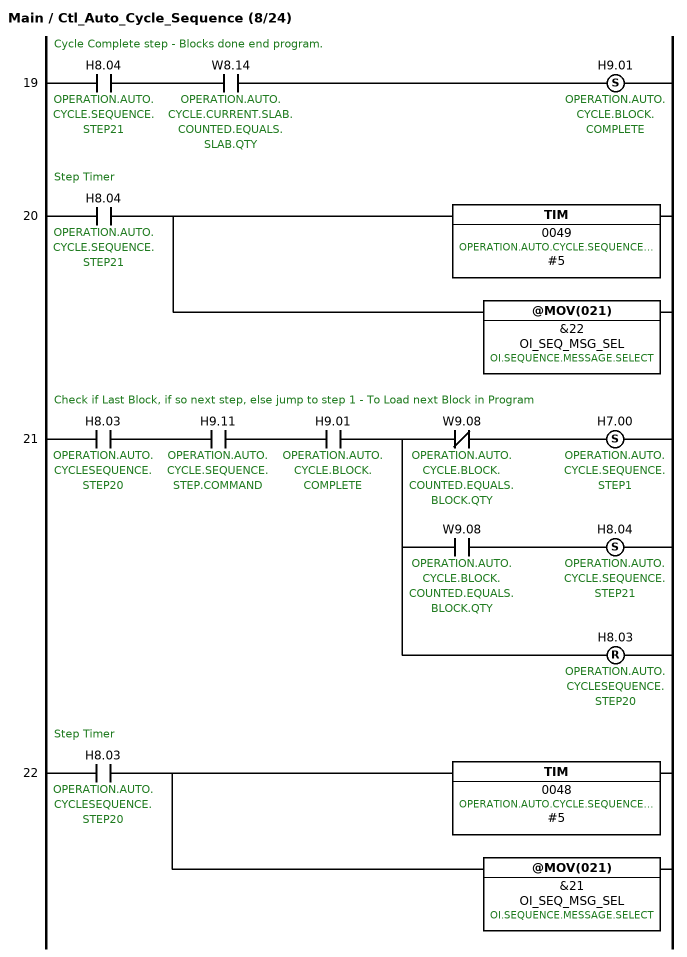
; [picture p24: Main / Ctl_Auto_Cycle_Sequence, rungs 19-22]
; rung 19: Cycle Complete step - Blocks done end program.
LD H8.04  ; OPERATION.AUTO.CYCLE.SEQUENCE.STEP21
AND W8.14  ; OPERATION.AUTO.CYCLE.CURRENT.SLAB.COUNTED.EQUALS.SLAB.QTY
SET H9.01  ; OPERATION.AUTO.CYCLE.BLOCK.COMPLETE
; rung 20: Step Timer
LD H8.04  ; OPERATION.AUTO.CYCLE.SEQUENCE.STEP21
TIM 0049 #5  ; OPERATION.AUTO.CYCLE.SEQUENCE.STEP21.TIMER
@MOV(021) &22 OI_SEQ_MSG_SEL  ; OI.SEQUENCE.MESSAGE.SELECT
; rung 21: Check if Last Block, if so next step, else jump to step 1 - To Load next Block in Program
LD H8.03  ; OPERATION.AUTO.CYCLESEQUENCE.STEP20
AND H9.11  ; OPERATION.AUTO.CYCLE.SEQUENCE.STEP.COMMAND
AND H9.01  ; OPERATION.AUTO.CYCLE.BLOCK.COMPLETE
OUT TR0
ANDNOT W9.08  ; OPERATION.AUTO.CYCLE.BLOCK.COUNTED.EQUALS.BLOCK.QTY
SET H7.00  ; OPERATION.AUTO.CYCLE.SEQUENCE.STEP1
LD TR0
AND W9.08  ; OPERATION.AUTO.CYCLE.BLOCK.COUNTED.EQUALS.BLOCK.QTY
SET H8.04  ; OPERATION.AUTO.CYCLE.SEQUENCE.STEP21
LD TR0
RSET H8.03  ; OPERATION.AUTO.CYCLESEQUENCE.STEP20
; rung 22: Step Timer
LD H8.03  ; OPERATION.AUTO.CYCLESEQUENCE.STEP20
TIM 0048 #5  ; OPERATION.AUTO.CYCLE.SEQUENCE.STEP20.TIMER
@MOV(021) &21 OI_SEQ_MSG_SEL  ; OI.SEQUENCE.MESSAGE.SELECT

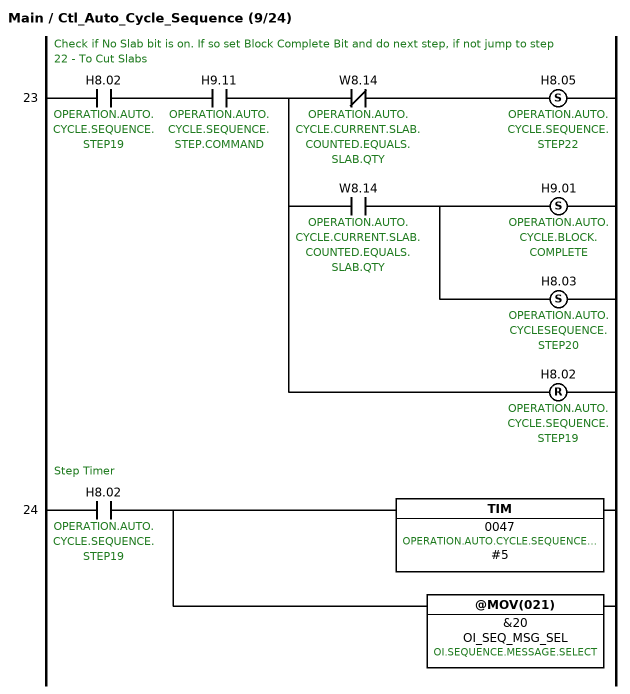
; rung 23: Check if No Slab bit is on. If so set Block Complete Bit and do next step, if not jump to step 22 - To Cut Slabs
LD H8.02  ; OPERATION.AUTO.CYCLE.SEQUENCE.STEP19
AND H9.11  ; OPERATION.AUTO.CYCLE.SEQUENCE.STEP.COMMAND
OUT TR0
ANDNOT W8.14  ; OPERATION.AUTO.CYCLE.CURRENT.SLAB.COUNTED.EQUALS.SLAB.QTY
SET H8.05  ; OPERATION.AUTO.CYCLE.SEQUENCE.STEP22
LD TR0
AND W8.14  ; OPERATION.AUTO.CYCLE.CURRENT.SLAB.COUNTED.EQUALS.SLAB.QTY
SET H9.01  ; OPERATION.AUTO.CYCLE.BLOCK.COMPLETE
SET H8.03  ; OPERATION.AUTO.CYCLESEQUENCE.STEP20
LD TR0
RSET H8.02  ; OPERATION.AUTO.CYCLE.SEQUENCE.STEP19
; rung 24: Step Timer
LD H8.02  ; OPERATION.AUTO.CYCLE.SEQUENCE.STEP19
TIM 0047 #5  ; OPERATION.AUTO.CYCLE.SEQUENCE.STEP19.TIMER
@MOV(021) &20 OI_SEQ_MSG_SEL  ; OI.SEQUENCE.MESSAGE.SELECT

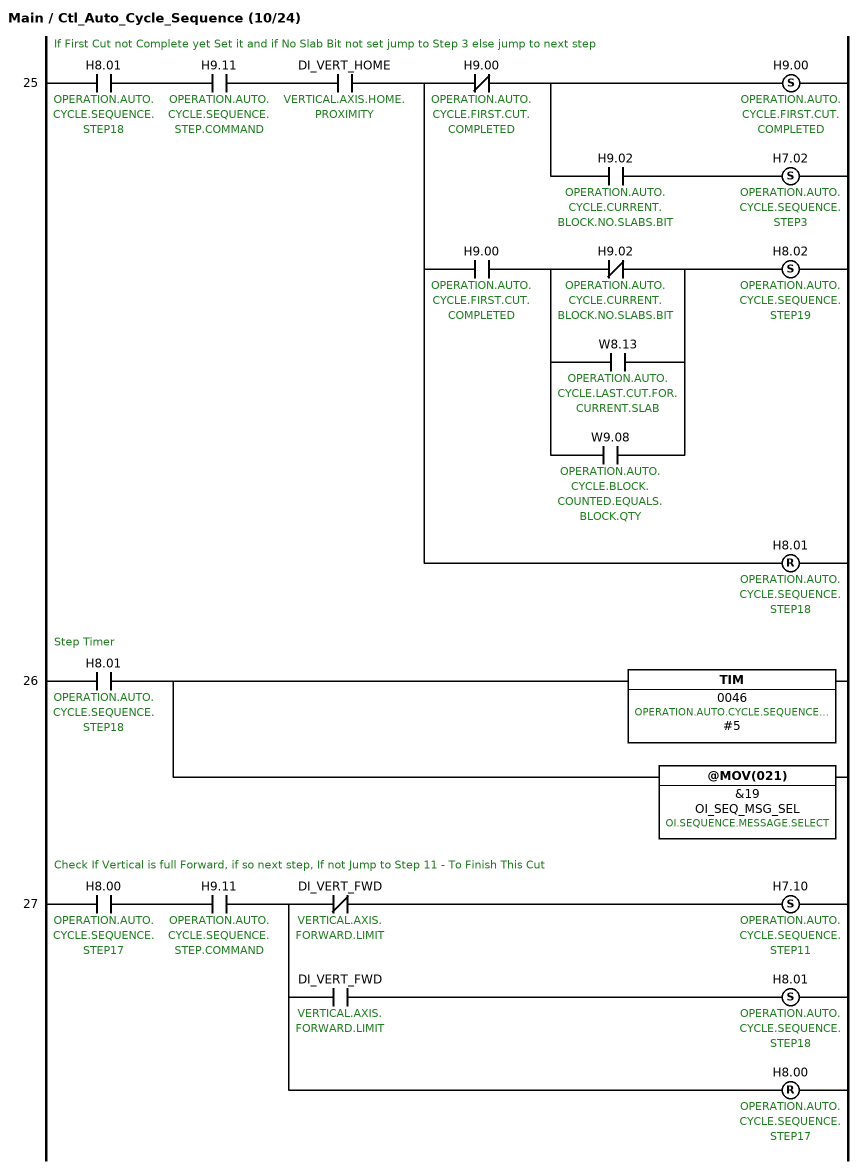
; rung 25: If First Cut not Complete yet Set it and if No Slab Bit not set jump to Step 3 else jump to next step
LD H8.01  ; OPERATION.AUTO.CYCLE.SEQUENCE.STEP18
AND H9.11  ; OPERATION.AUTO.CYCLE.SEQUENCE.STEP.COMMAND
AND DI_VERT_HOME  ; VERTICAL.AXIS.HOME.PROXIMITY
OUT TR0
ANDNOT H9.00  ; OPERATION.AUTO.CYCLE.FIRST.CUT.COMPLETED
SET H9.00  ; OPERATION.AUTO.CYCLE.FIRST.CUT.COMPLETED
AND H9.02  ; OPERATION.AUTO.CYCLE.CURRENT.BLOCK.NO.SLABS.BIT
SET H7.02  ; OPERATION.AUTO.CYCLE.SEQUENCE.STEP3
LD TR0
AND H9.00  ; OPERATION.AUTO.CYCLE.FIRST.CUT.COMPLETED
LDNOT H9.02  ; OPERATION.AUTO.CYCLE.CURRENT.BLOCK.NO.SLABS.BIT
OR W8.13  ; OPERATION.AUTO.CYCLE.LAST.CUT.FOR.CURRENT.SLAB
OR W9.08  ; OPERATION.AUTO.CYCLE.BLOCK.COUNTED.EQUALS.BLOCK.QTY
ANDLD
SET H8.02  ; OPERATION.AUTO.CYCLE.SEQUENCE.STEP19
LD TR0
RSET H8.01  ; OPERATION.AUTO.CYCLE.SEQUENCE.STEP18
; rung 26: Step Timer
LD H8.01  ; OPERATION.AUTO.CYCLE.SEQUENCE.STEP18
TIM 0046 #5  ; OPERATION.AUTO.CYCLE.SEQUENCE.STEP18.TIMER
@MOV(021) &19 OI_SEQ_MSG_SEL  ; OI.SEQUENCE.MESSAGE.SELECT
; rung 27: Check If Vertical is full Forward, if so next step, If not Jump to Step 11 - To Finish This Cut
LD H8.00  ; OPERATION.AUTO.CYCLE.SEQUENCE.STEP17
AND H9.11  ; OPERATION.AUTO.CYCLE.SEQUENCE.STEP.COMMAND
OUT TR0
ANDNOT DI_VERT_FWD  ; VERTICAL.AXIS.FORWARD.LIMIT
SET H7.10  ; OPERATION.AUTO.CYCLE.SEQUENCE.STEP11
LD TR0
AND DI_VERT_FWD  ; VERTICAL.AXIS.FORWARD.LIMIT
SET H8.01  ; OPERATION.AUTO.CYCLE.SEQUENCE.STEP18
LD TR0
RSET H8.00  ; OPERATION.AUTO.CYCLE.SEQUENCE.STEP17

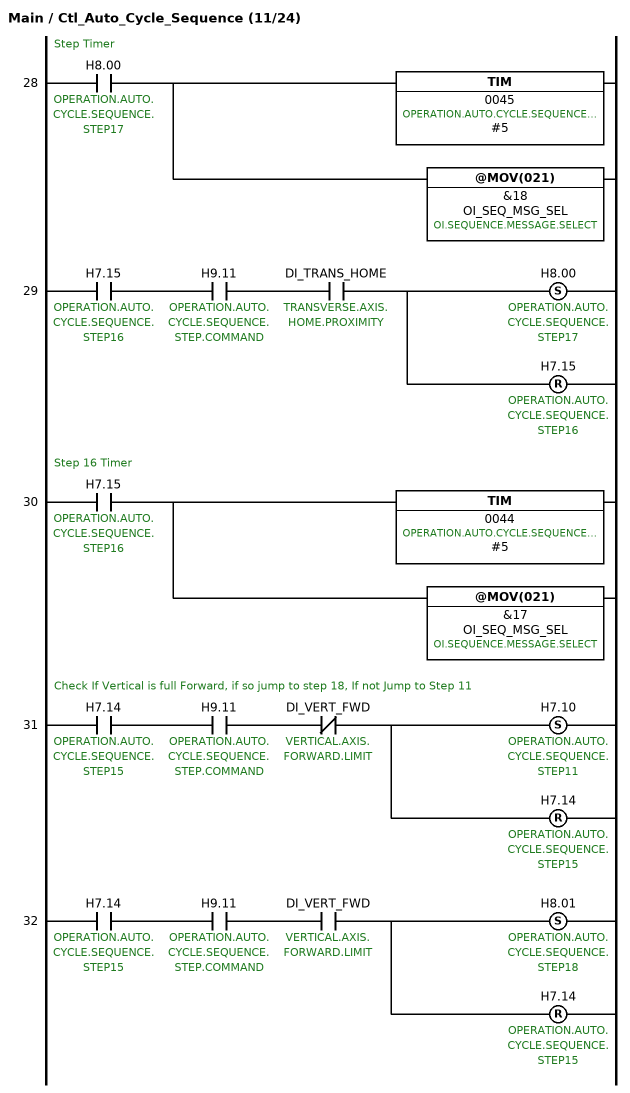
; rung 28: Step Timer
LD H8.00  ; OPERATION.AUTO.CYCLE.SEQUENCE.STEP17
TIM 0045 #5  ; OPERATION.AUTO.CYCLE.SEQUENCE.STEP17.TIMER
@MOV(021) &18 OI_SEQ_MSG_SEL  ; OI.SEQUENCE.MESSAGE.SELECT
; rung 29
LD H7.15  ; OPERATION.AUTO.CYCLE.SEQUENCE.STEP16
AND H9.11  ; OPERATION.AUTO.CYCLE.SEQUENCE.STEP.COMMAND
AND DI_TRANS_HOME  ; TRANSVERSE.AXIS.HOME.PROXIMITY
SET H8.00  ; OPERATION.AUTO.CYCLE.SEQUENCE.STEP17
RSET H7.15  ; OPERATION.AUTO.CYCLE.SEQUENCE.STEP16
; rung 30: Step 16 Timer
LD H7.15  ; OPERATION.AUTO.CYCLE.SEQUENCE.STEP16
TIM 0044 #5  ; OPERATION.AUTO.CYCLE.SEQUENCE.STEP16.TIMER
@MOV(021) &17 OI_SEQ_MSG_SEL  ; OI.SEQUENCE.MESSAGE.SELECT
; rung 31: Check If Vertical is full Forward, if so jump to step 18, If not Jump to Step 11
LD H7.14  ; OPERATION.AUTO.CYCLE.SEQUENCE.STEP15
AND H9.11  ; OPERATION.AUTO.CYCLE.SEQUENCE.STEP.COMMAND
ANDNOT DI_VERT_FWD  ; VERTICAL.AXIS.FORWARD.LIMIT
SET H7.10  ; OPERATION.AUTO.CYCLE.SEQUENCE.STEP11
RSET H7.14  ; OPERATION.AUTO.CYCLE.SEQUENCE.STEP15
; rung 32
LD H7.14  ; OPERATION.AUTO.CYCLE.SEQUENCE.STEP15
AND H9.11  ; OPERATION.AUTO.CYCLE.SEQUENCE.STEP.COMMAND
AND DI_VERT_FWD  ; VERTICAL.AXIS.FORWARD.LIMIT
SET H8.01  ; OPERATION.AUTO.CYCLE.SEQUENCE.STEP18
RSET H7.14  ; OPERATION.AUTO.CYCLE.SEQUENCE.STEP15

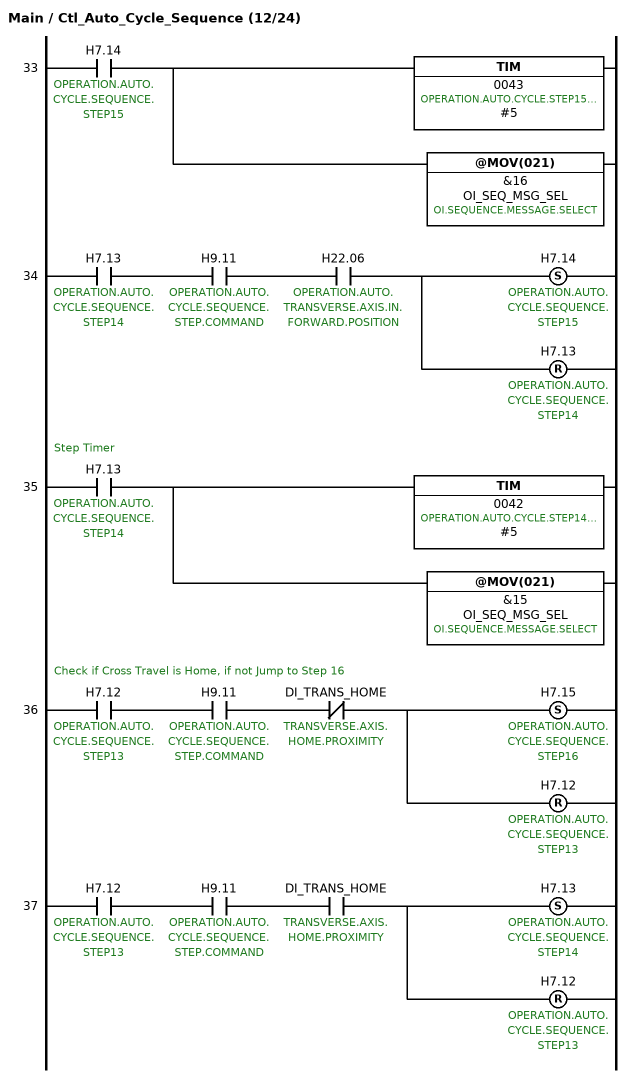
; rung 33
LD H7.14  ; OPERATION.AUTO.CYCLE.SEQUENCE.STEP15
TIM 0043 #5  ; OPERATION.AUTO.CYCLE.STEP15.TIMER
@MOV(021) &16 OI_SEQ_MSG_SEL  ; OI.SEQUENCE.MESSAGE.SELECT
; rung 34
LD H7.13  ; OPERATION.AUTO.CYCLE.SEQUENCE.STEP14
AND H9.11  ; OPERATION.AUTO.CYCLE.SEQUENCE.STEP.COMMAND
AND H22.06  ; OPERATION.AUTO.TRANSVERSE.AXIS.IN.FORWARD.POSITION
SET H7.14  ; OPERATION.AUTO.CYCLE.SEQUENCE.STEP15
RSET H7.13  ; OPERATION.AUTO.CYCLE.SEQUENCE.STEP14
; rung 35: Step Timer
LD H7.13  ; OPERATION.AUTO.CYCLE.SEQUENCE.STEP14
TIM 0042 #5  ; OPERATION.AUTO.CYCLE.STEP14.TIMER
@MOV(021) &15 OI_SEQ_MSG_SEL  ; OI.SEQUENCE.MESSAGE.SELECT
; rung 36: Check if Cross Travel is Home, if not Jump to Step 16
LD H7.12  ; OPERATION.AUTO.CYCLE.SEQUENCE.STEP13
AND H9.11  ; OPERATION.AUTO.CYCLE.SEQUENCE.STEP.COMMAND
ANDNOT DI_TRANS_HOME  ; TRANSVERSE.AXIS.HOME.PROXIMITY
SET H7.15  ; OPERATION.AUTO.CYCLE.SEQUENCE.STEP16
RSET H7.12  ; OPERATION.AUTO.CYCLE.SEQUENCE.STEP13
; rung 37
LD H7.12  ; OPERATION.AUTO.CYCLE.SEQUENCE.STEP13
AND H9.11  ; OPERATION.AUTO.CYCLE.SEQUENCE.STEP.COMMAND
AND DI_TRANS_HOME  ; TRANSVERSE.AXIS.HOME.PROXIMITY
SET H7.13  ; OPERATION.AUTO.CYCLE.SEQUENCE.STEP14
RSET H7.12  ; OPERATION.AUTO.CYCLE.SEQUENCE.STEP13

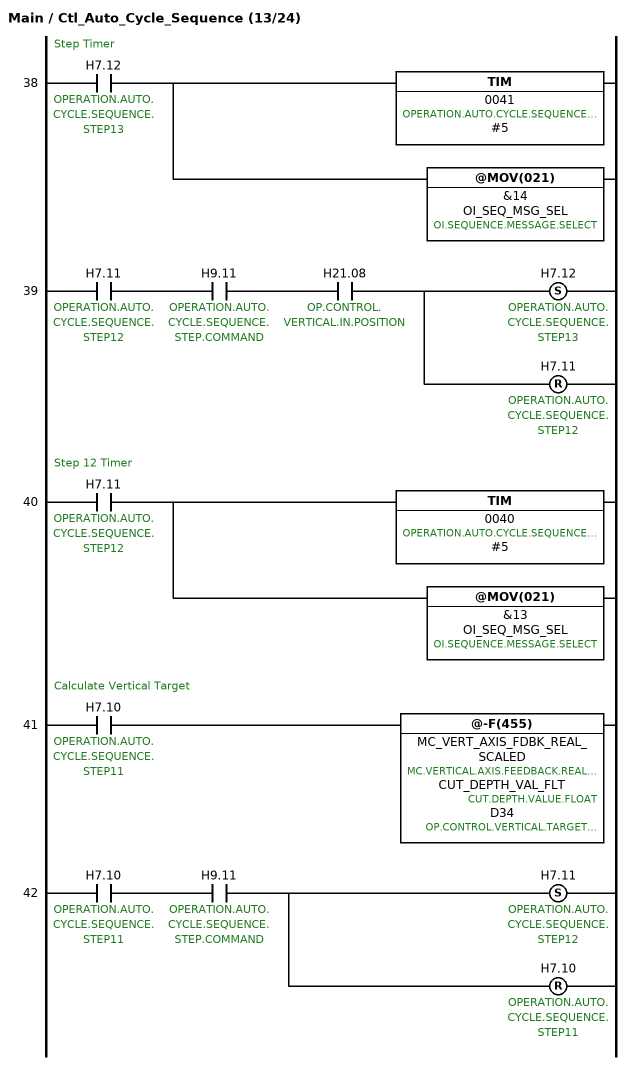
; rung 38: Step Timer
LD H7.12  ; OPERATION.AUTO.CYCLE.SEQUENCE.STEP13
TIM 0041 #5  ; OPERATION.AUTO.CYCLE.SEQUENCE.STEP13.TIME
@MOV(021) &14 OI_SEQ_MSG_SEL  ; OI.SEQUENCE.MESSAGE.SELECT
; rung 39
LD H7.11  ; OPERATION.AUTO.CYCLE.SEQUENCE.STEP12
AND H9.11  ; OPERATION.AUTO.CYCLE.SEQUENCE.STEP.COMMAND
AND H21.08  ; OP.CONTROL.VERTICAL.IN.POSITION
SET H7.12  ; OPERATION.AUTO.CYCLE.SEQUENCE.STEP13
RSET H7.11  ; OPERATION.AUTO.CYCLE.SEQUENCE.STEP12
; rung 40: Step 12 Timer
LD H7.11  ; OPERATION.AUTO.CYCLE.SEQUENCE.STEP12
TIM 0040 #5  ; OPERATION.AUTO.CYCLE.SEQUENCE.STEP12.TIMER
@MOV(021) &13 OI_SEQ_MSG_SEL  ; OI.SEQUENCE.MESSAGE.SELECT
; rung 41: Calculate Vertical Target
LD H7.10  ; OPERATION.AUTO.CYCLE.SEQUENCE.STEP11
@-F(455) MC_VERT_AXIS_FDBK_REAL_SCALED CUT_DEPTH_VAL_FLT D34  ; MC.VERTICAL.AXIS.FEEDBACK.REAL.SCALED.INCH, CUT.DEPTH.VALUE.FLOAT, OP.CONTROL.VERTICAL.TARGET.SCALED
; rung 42
LD H7.10  ; OPERATION.AUTO.CYCLE.SEQUENCE.STEP11
AND H9.11  ; OPERATION.AUTO.CYCLE.SEQUENCE.STEP.COMMAND
SET H7.11  ; OPERATION.AUTO.CYCLE.SEQUENCE.STEP12
RSET H7.10  ; OPERATION.AUTO.CYCLE.SEQUENCE.STEP11

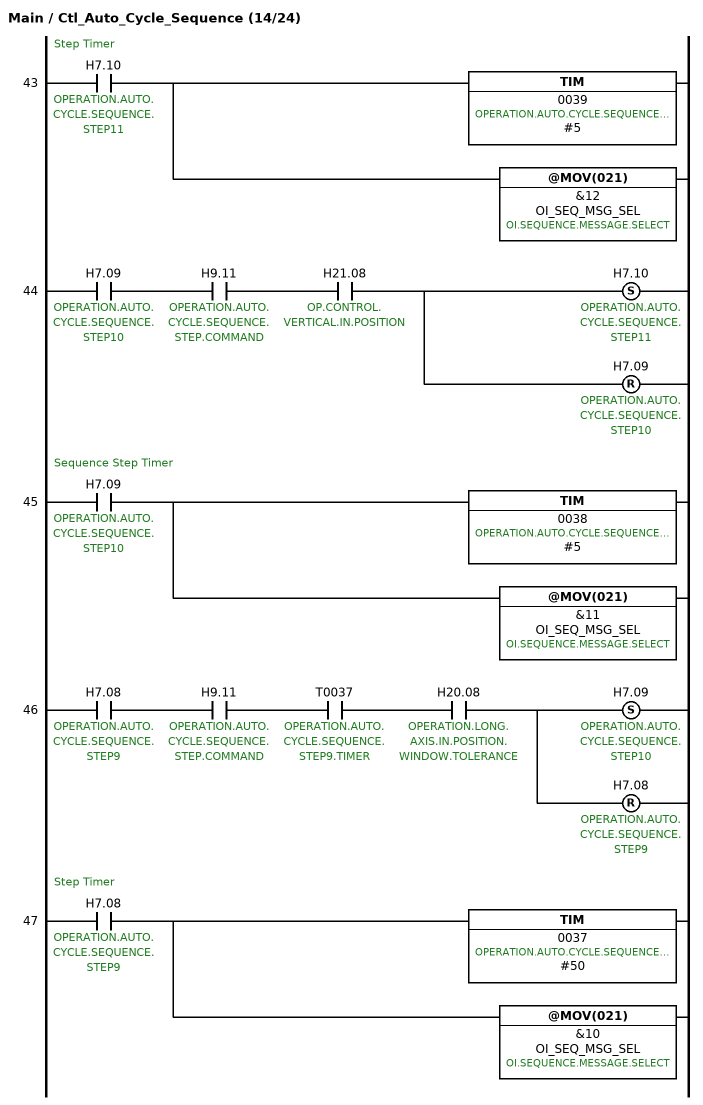
; rung 43: Step Timer
LD H7.10  ; OPERATION.AUTO.CYCLE.SEQUENCE.STEP11
TIM 0039 #5  ; OPERATION.AUTO.CYCLE.SEQUENCE.STEP11.TIMER
@MOV(021) &12 OI_SEQ_MSG_SEL  ; OI.SEQUENCE.MESSAGE.SELECT
; rung 44
LD H7.09  ; OPERATION.AUTO.CYCLE.SEQUENCE.STEP10
AND H9.11  ; OPERATION.AUTO.CYCLE.SEQUENCE.STEP.COMMAND
AND H21.08  ; OP.CONTROL.VERTICAL.IN.POSITION
SET H7.10  ; OPERATION.AUTO.CYCLE.SEQUENCE.STEP11
RSET H7.09  ; OPERATION.AUTO.CYCLE.SEQUENCE.STEP10
; rung 45: Sequence Step Timer
LD H7.09  ; OPERATION.AUTO.CYCLE.SEQUENCE.STEP10
TIM 0038 #5  ; OPERATION.AUTO.CYCLE.SEQUENCE.STEP10.TIMER
@MOV(021) &11 OI_SEQ_MSG_SEL  ; OI.SEQUENCE.MESSAGE.SELECT
; rung 46
LD H7.08  ; OPERATION.AUTO.CYCLE.SEQUENCE.STEP9
AND H9.11  ; OPERATION.AUTO.CYCLE.SEQUENCE.STEP.COMMAND
AND T0037  ; OPERATION.AUTO.CYCLE.SEQUENCE.STEP9.TIMER
AND H20.08  ; OPERATION.LONG.AXIS.IN.POSITION.WINDOW.TOLERANCE
SET H7.09  ; OPERATION.AUTO.CYCLE.SEQUENCE.STEP10
RSET H7.08  ; OPERATION.AUTO.CYCLE.SEQUENCE.STEP9
; rung 47: Step Timer
LD H7.08  ; OPERATION.AUTO.CYCLE.SEQUENCE.STEP9
TIM 0037 #50  ; OPERATION.AUTO.CYCLE.SEQUENCE.STEP9.TIMER
@MOV(021) &10 OI_SEQ_MSG_SEL  ; OI.SEQUENCE.MESSAGE.SELECT

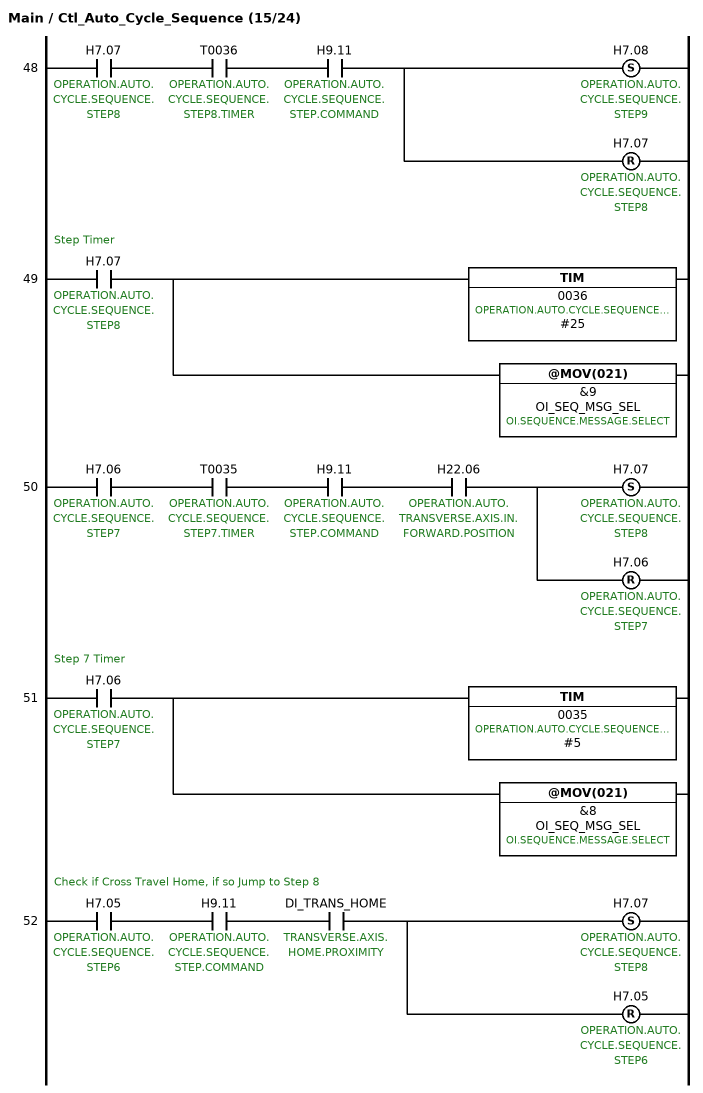
; rung 48
LD H7.07  ; OPERATION.AUTO.CYCLE.SEQUENCE.STEP8
AND T0036  ; OPERATION.AUTO.CYCLE.SEQUENCE.STEP8.TIMER
AND H9.11  ; OPERATION.AUTO.CYCLE.SEQUENCE.STEP.COMMAND
SET H7.08  ; OPERATION.AUTO.CYCLE.SEQUENCE.STEP9
RSET H7.07  ; OPERATION.AUTO.CYCLE.SEQUENCE.STEP8
; rung 49: Step Timer
LD H7.07  ; OPERATION.AUTO.CYCLE.SEQUENCE.STEP8
TIM 0036 #25  ; OPERATION.AUTO.CYCLE.SEQUENCE.STEP8.TIMER
@MOV(021) &9 OI_SEQ_MSG_SEL  ; OI.SEQUENCE.MESSAGE.SELECT
; rung 50
LD H7.06  ; OPERATION.AUTO.CYCLE.SEQUENCE.STEP7
AND T0035  ; OPERATION.AUTO.CYCLE.SEQUENCE.STEP7.TIMER
AND H9.11  ; OPERATION.AUTO.CYCLE.SEQUENCE.STEP.COMMAND
AND H22.06  ; OPERATION.AUTO.TRANSVERSE.AXIS.IN.FORWARD.POSITION
SET H7.07  ; OPERATION.AUTO.CYCLE.SEQUENCE.STEP8
RSET H7.06  ; OPERATION.AUTO.CYCLE.SEQUENCE.STEP7
; rung 51: Step 7 Timer
LD H7.06  ; OPERATION.AUTO.CYCLE.SEQUENCE.STEP7
TIM 0035 #5  ; OPERATION.AUTO.CYCLE.SEQUENCE.STEP7.TIMER
@MOV(021) &8 OI_SEQ_MSG_SEL  ; OI.SEQUENCE.MESSAGE.SELECT
; rung 52: Check if Cross Travel Home, if so Jump to Step 8
LD H7.05  ; OPERATION.AUTO.CYCLE.SEQUENCE.STEP6
AND H9.11  ; OPERATION.AUTO.CYCLE.SEQUENCE.STEP.COMMAND
AND DI_TRANS_HOME  ; TRANSVERSE.AXIS.HOME.PROXIMITY
SET H7.07  ; OPERATION.AUTO.CYCLE.SEQUENCE.STEP8
RSET H7.05  ; OPERATION.AUTO.CYCLE.SEQUENCE.STEP6

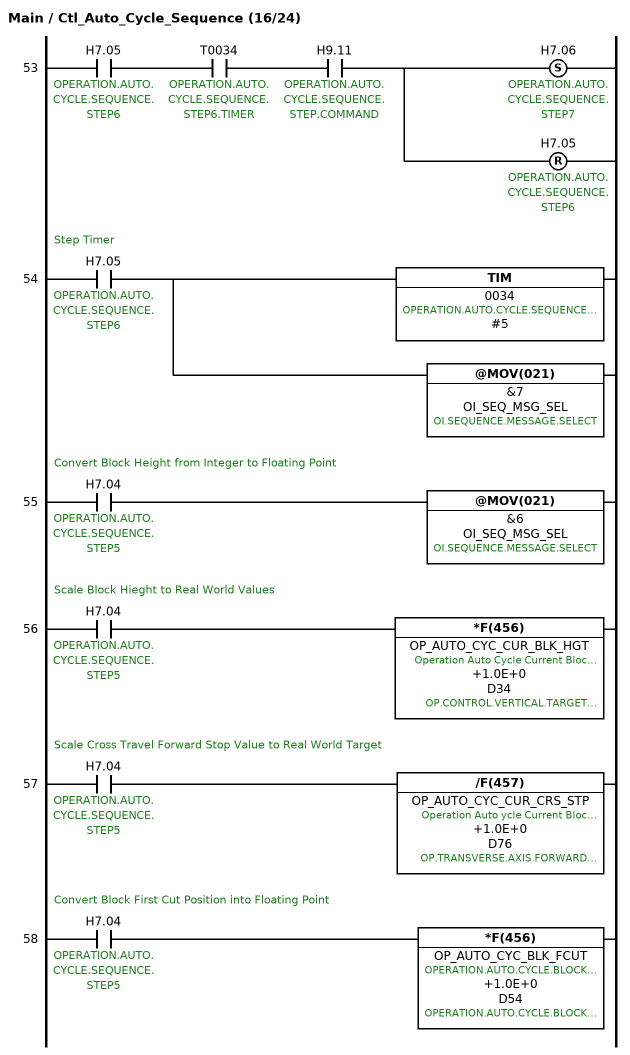
; rung 53
LD H7.05  ; OPERATION.AUTO.CYCLE.SEQUENCE.STEP6
AND T0034  ; OPERATION.AUTO.CYCLE.SEQUENCE.STEP6.TIMER
AND H9.11  ; OPERATION.AUTO.CYCLE.SEQUENCE.STEP.COMMAND
SET H7.06  ; OPERATION.AUTO.CYCLE.SEQUENCE.STEP7
RSET H7.05  ; OPERATION.AUTO.CYCLE.SEQUENCE.STEP6
; rung 54: Step Timer
LD H7.05  ; OPERATION.AUTO.CYCLE.SEQUENCE.STEP6
TIM 0034 #5  ; OPERATION.AUTO.CYCLE.SEQUENCE.STEP6.TIMER
@MOV(021) &7 OI_SEQ_MSG_SEL  ; OI.SEQUENCE.MESSAGE.SELECT
; rung 55: Convert Block Height from Integer to Floating Point
LD H7.04  ; OPERATION.AUTO.CYCLE.SEQUENCE.STEP5
@MOV(021) &6 OI_SEQ_MSG_SEL  ; OI.SEQUENCE.MESSAGE.SELECT
; rung 56: Scale Block Hieght to Real World Values
LD H7.04  ; OPERATION.AUTO.CYCLE.SEQUENCE.STEP5
*F(456) OP_AUTO_CYC_CUR_BLK_HGT +1.0E+0 D34  ; Operation Auto Cycle Current Block Height, OP.CONTROL.VERTICAL.TARGET.SCALED
; rung 57: Scale Cross Travel Forward Stop Value to Real World Target
LD H7.04  ; OPERATION.AUTO.CYCLE.SEQUENCE.STEP5
/F(457) OP_AUTO_CYC_CUR_CRS_STP +1.0E+0 D76  ; Operation Auto ycle Current Block Cross Stop, OP.TRANSVERSE.AXIS.FORWARD.TARGET
; rung 58: Convert Block First Cut Position into Floating Point
LD H7.04  ; OPERATION.AUTO.CYCLE.SEQUENCE.STEP5
*F(456) OP_AUTO_CYC_BLK_FCUT +1.0E+0 D54  ; OPERATION.AUTO.CYCLE.BLOCK.FIRST.CUT.WORKING, OPERATION.AUTO.CYCLE.BLOCK.FIRST.CUT.REAL

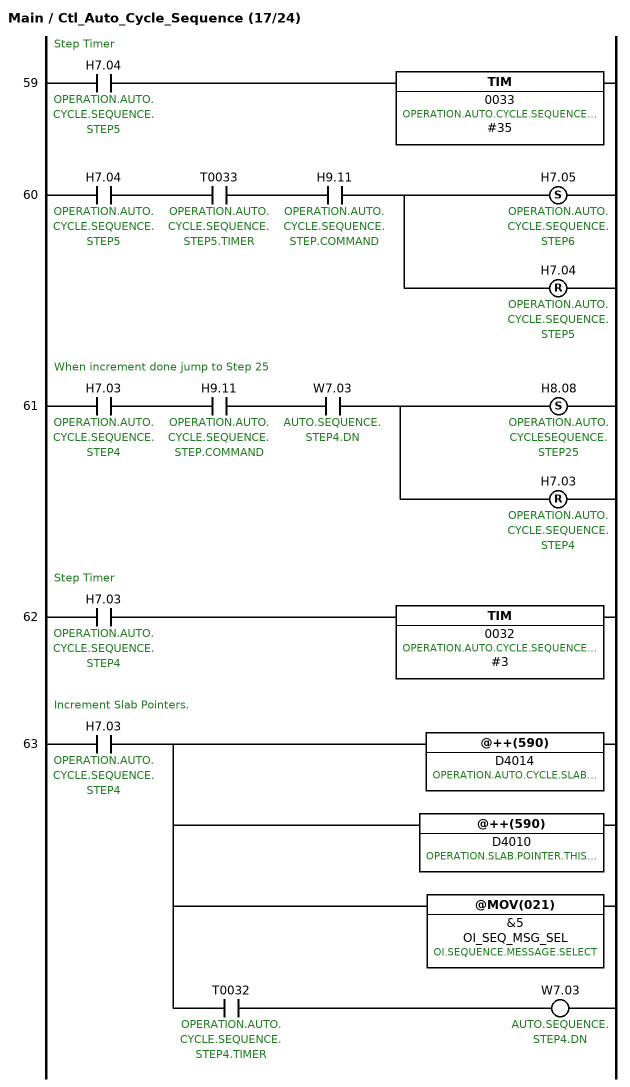
; rung 59: Step Timer
LD H7.04  ; OPERATION.AUTO.CYCLE.SEQUENCE.STEP5
TIM 0033 #35  ; OPERATION.AUTO.CYCLE.SEQUENCE.STEP5.TIMER
; rung 60
LD H7.04  ; OPERATION.AUTO.CYCLE.SEQUENCE.STEP5
AND T0033  ; OPERATION.AUTO.CYCLE.SEQUENCE.STEP5.TIMER
AND H9.11  ; OPERATION.AUTO.CYCLE.SEQUENCE.STEP.COMMAND
SET H7.05  ; OPERATION.AUTO.CYCLE.SEQUENCE.STEP6
RSET H7.04  ; OPERATION.AUTO.CYCLE.SEQUENCE.STEP5
; rung 61: When increment done jump to Step 25
LD H7.03  ; OPERATION.AUTO.CYCLE.SEQUENCE.STEP4
AND H9.11  ; OPERATION.AUTO.CYCLE.SEQUENCE.STEP.COMMAND
AND W7.03  ; AUTO.SEQUENCE.STEP4.DN
SET H8.08  ; OPERATION.AUTO.CYCLESEQUENCE.STEP25
RSET H7.03  ; OPERATION.AUTO.CYCLE.SEQUENCE.STEP4
; rung 62: Step Timer
LD H7.03  ; OPERATION.AUTO.CYCLE.SEQUENCE.STEP4
TIM 0032 #3  ; OPERATION.AUTO.CYCLE.SEQUENCE.STEP4.TIMER
; rung 63: Increment Slab Pointers.
LD H7.03  ; OPERATION.AUTO.CYCLE.SEQUENCE.STEP4
@++(590) D4014  ; OPERATION.AUTO.CYCLE.SLAB.POINTER
@++(590) D4010  ; OPERATION.SLAB.POINTER.THIS.BLOCK
@MOV(021) &5 OI_SEQ_MSG_SEL  ; OI.SEQUENCE.MESSAGE.SELECT
AND T0032  ; OPERATION.AUTO.CYCLE.SEQUENCE.STEP4.TIMER
OUT W7.03  ; AUTO.SEQUENCE.STEP4.DN

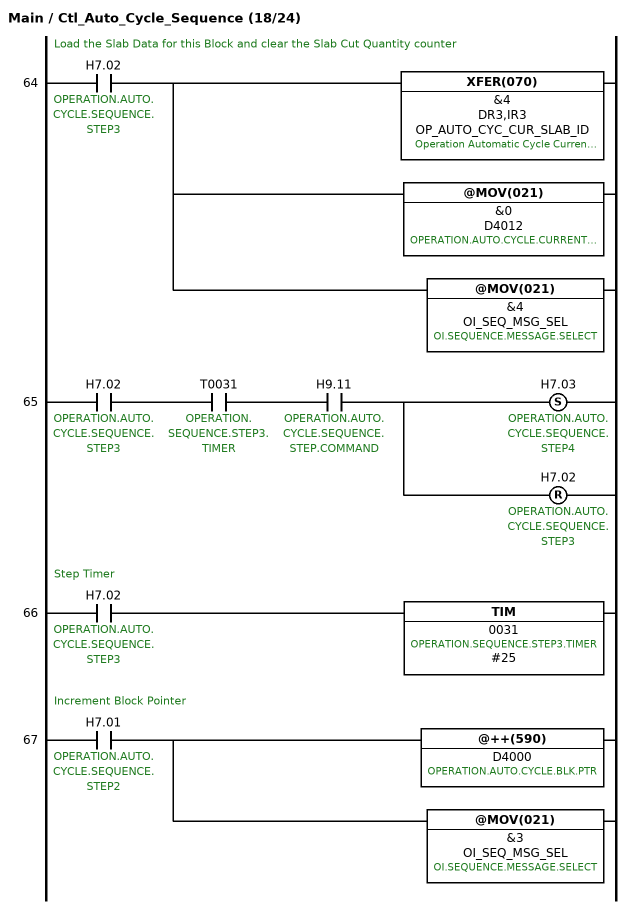
; rung 64: Load the Slab Data for this Block and clear the Slab Cut Quantity counter
LD H7.02  ; OPERATION.AUTO.CYCLE.SEQUENCE.STEP3
XFER(070) &4 DR3,IR3 OP_AUTO_CYC_CUR_SLAB_ID  ; Operation Automatic Cycle Current Slab ID
@MOV(021) &0 D4012  ; OPERATION.AUTO.CYCLE.CURRENT.SLAB.CUT.COUNTER
@MOV(021) &4 OI_SEQ_MSG_SEL  ; OI.SEQUENCE.MESSAGE.SELECT
; rung 65
LD H7.02  ; OPERATION.AUTO.CYCLE.SEQUENCE.STEP3
AND T0031  ; OPERATION.SEQUENCE.STEP3.TIMER
AND H9.11  ; OPERATION.AUTO.CYCLE.SEQUENCE.STEP.COMMAND
SET H7.03  ; OPERATION.AUTO.CYCLE.SEQUENCE.STEP4
RSET H7.02  ; OPERATION.AUTO.CYCLE.SEQUENCE.STEP3
; rung 66: Step Timer
LD H7.02  ; OPERATION.AUTO.CYCLE.SEQUENCE.STEP3
TIM 0031 #25  ; OPERATION.SEQUENCE.STEP3.TIMER
; rung 67: Increment Block Pointer
LD H7.01  ; OPERATION.AUTO.CYCLE.SEQUENCE.STEP2
@++(590) D4000  ; OPERATION.AUTO.CYCLE.BLK.PTR
@MOV(021) &3 OI_SEQ_MSG_SEL  ; OI.SEQUENCE.MESSAGE.SELECT

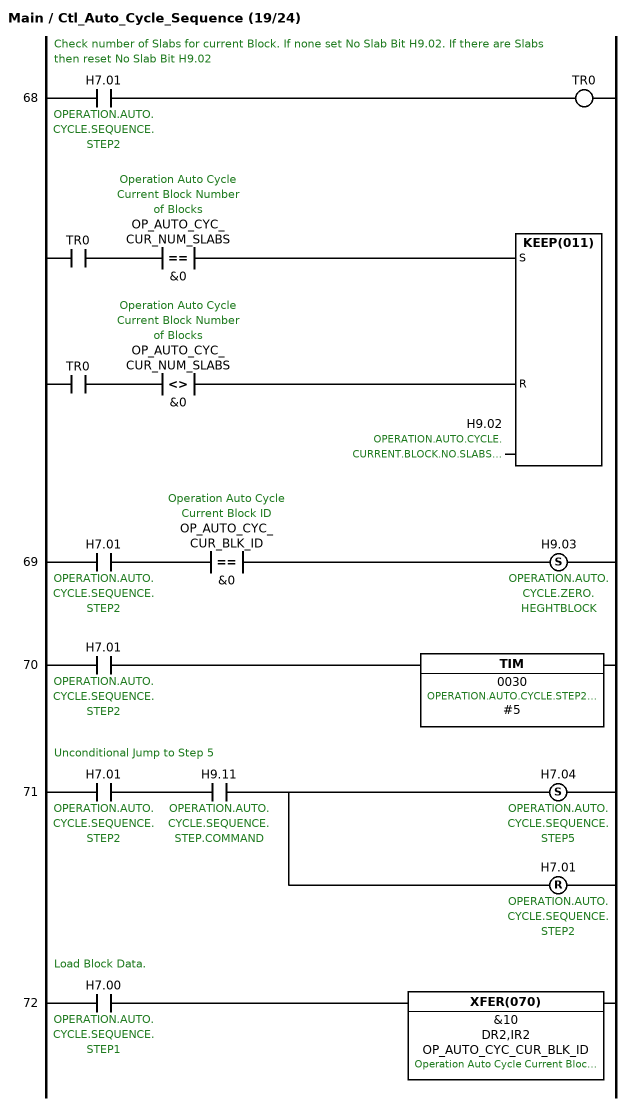
; rung 68: Check number of Slabs for current Block. If none set No Slab Bit H9.02. If there are Slabs then reset No Slab Bit H9.02
LD H7.01  ; OPERATION.AUTO.CYCLE.SEQUENCE.STEP2
OUT TR0
AND=(300) OP_AUTO_CYC_CUR_NUM_SLABS &0  ; Operation Auto Cycle Current Block Number of Blocks
LD TR0
AND<>(305) OP_AUTO_CYC_CUR_NUM_SLABS &0  ; Operation Auto Cycle Current Block Number of Blocks
KEEP(011) H9.02  ; OPERATION.AUTO.CYCLE.CURRENT.BLOCK.NO.SLABS.BIT
; rung 69
LD H7.01  ; OPERATION.AUTO.CYCLE.SEQUENCE.STEP2
AND=(300) OP_AUTO_CYC_CUR_BLK_ID &0  ; Operation Auto Cycle Current Block ID
SET H9.03  ; OPERATION.AUTO.CYCLE.ZERO.HEGHTBLOCK
; rung 70
LD H7.01  ; OPERATION.AUTO.CYCLE.SEQUENCE.STEP2
TIM 0030 #5  ; OPERATION.AUTO.CYCLE.STEP2.TIMER
; rung 71: Unconditional Jump to Step 5
LD H7.01  ; OPERATION.AUTO.CYCLE.SEQUENCE.STEP2
AND H9.11  ; OPERATION.AUTO.CYCLE.SEQUENCE.STEP.COMMAND
SET H7.04  ; OPERATION.AUTO.CYCLE.SEQUENCE.STEP5
RSET H7.01  ; OPERATION.AUTO.CYCLE.SEQUENCE.STEP2
; rung 72: Load Block Data.
LD H7.00  ; OPERATION.AUTO.CYCLE.SEQUENCE.STEP1
XFER(070) &10 DR2,IR2 OP_AUTO_CYC_CUR_BLK_ID  ; Operation Auto Cycle Current Block ID

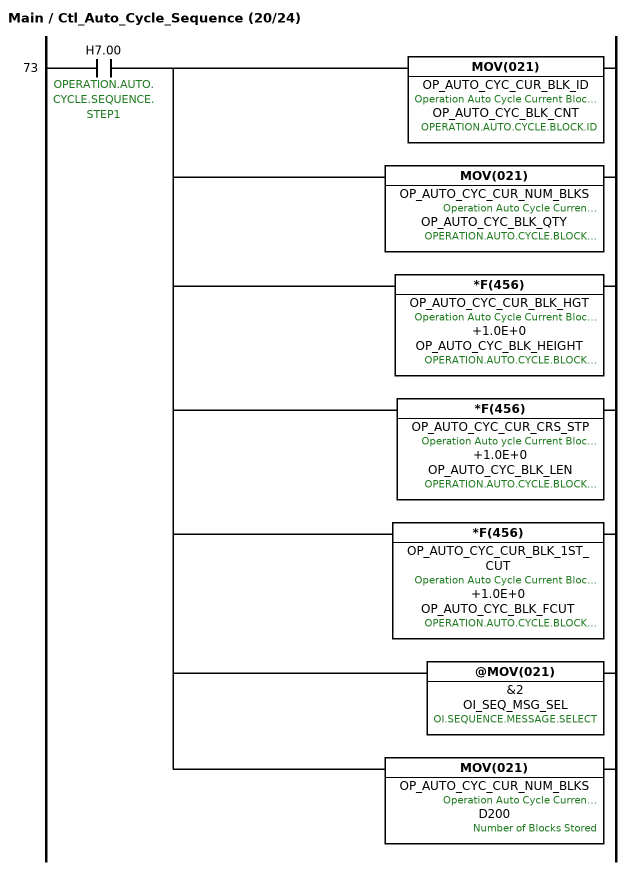
; rung 73
LD H7.00  ; OPERATION.AUTO.CYCLE.SEQUENCE.STEP1
MOV(021) OP_AUTO_CYC_CUR_BLK_ID OP_AUTO_CYC_BLK_CNT  ; Operation Auto Cycle Current Block ID, OPERATION.AUTO.CYCLE.BLOCK.ID
MOV(021) OP_AUTO_CYC_CUR_NUM_BLKS OP_AUTO_CYC_BLK_QTY  ; Operation Auto Cycle Current Number of Blocks, OPERATION.AUTO.CYCLE.BLOCK.QUANTITY
*F(456) OP_AUTO_CYC_CUR_BLK_HGT +1.0E+0 OP_AUTO_CYC_BLK_HEIGHT  ; Operation Auto Cycle Current Block Height, OPERATION.AUTO.CYCLE.BLOCK.HEIGHT.WORKING
*F(456) OP_AUTO_CYC_CUR_CRS_STP +1.0E+0 OP_AUTO_CYC_BLK_LEN  ; Operation Auto ycle Current Block Cross Stop, OPERATION.AUTO.CYCLE.BLOCK.TRANSVERSE.AXIS.STOP.POSITION.WORKING
*F(456) OP_AUTO_CYC_CUR_BLK_1ST_CUT +1.0E+0 OP_AUTO_CYC_BLK_FCUT  ; Operation Auto Cycle Current Block First Cut Location, OPERATION.AUTO.CYCLE.BLOCK.FIRST.CUT.WORKING
@MOV(021) &2 OI_SEQ_MSG_SEL  ; OI.SEQUENCE.MESSAGE.SELECT
MOV(021) OP_AUTO_CYC_CUR_NUM_BLKS D200  ; Operation Auto Cycle Current Number of Blocks, Number of Blocks Stored

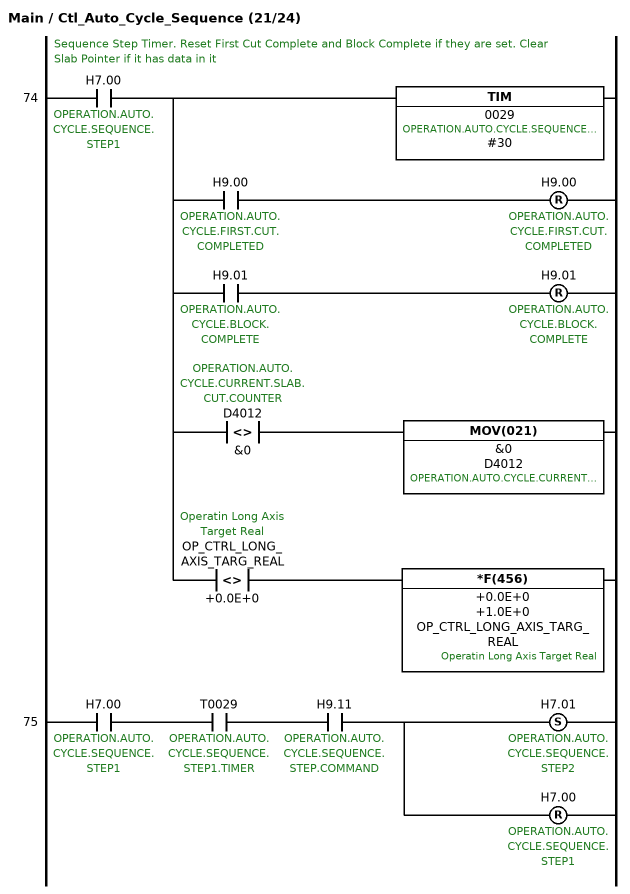
; rung 74: Sequence Step Timer. Reset First Cut Complete and Block Complete if they are set. Clear Slab Pointer if it has data in it
LD H7.00  ; OPERATION.AUTO.CYCLE.SEQUENCE.STEP1
OUT TR0
TIM 0029 #30  ; OPERATION.AUTO.CYCLE.SEQUENCE.STEP1.TIMER
AND H9.00  ; OPERATION.AUTO.CYCLE.FIRST.CUT.COMPLETED
RSET H9.00  ; OPERATION.AUTO.CYCLE.FIRST.CUT.COMPLETED
LD TR0
AND H9.01  ; OPERATION.AUTO.CYCLE.BLOCK.COMPLETE
RSET H9.01  ; OPERATION.AUTO.CYCLE.BLOCK.COMPLETE
LD TR0
AND<>(305) D4012 &0  ; OPERATION.AUTO.CYCLE.CURRENT.SLAB.CUT.COUNTER
MOV(021) &0 D4012  ; OPERATION.AUTO.CYCLE.CURRENT.SLAB.CUT.COUNTER
LD TR0
AND<>F(330) OP_CTRL_LONG_AXIS_TARG_REAL +0.0E+0  ; Operatin Long Axis Target Real
*F(456) +0.0E+0 +1.0E+0 OP_CTRL_LONG_AXIS_TARG_REAL  ; Operatin Long Axis Target Real
; rung 75
LD H7.00  ; OPERATION.AUTO.CYCLE.SEQUENCE.STEP1
AND T0029  ; OPERATION.AUTO.CYCLE.SEQUENCE.STEP1.TIMER
AND H9.11  ; OPERATION.AUTO.CYCLE.SEQUENCE.STEP.COMMAND
SET H7.01  ; OPERATION.AUTO.CYCLE.SEQUENCE.STEP2
RSET H7.00  ; OPERATION.AUTO.CYCLE.SEQUENCE.STEP1

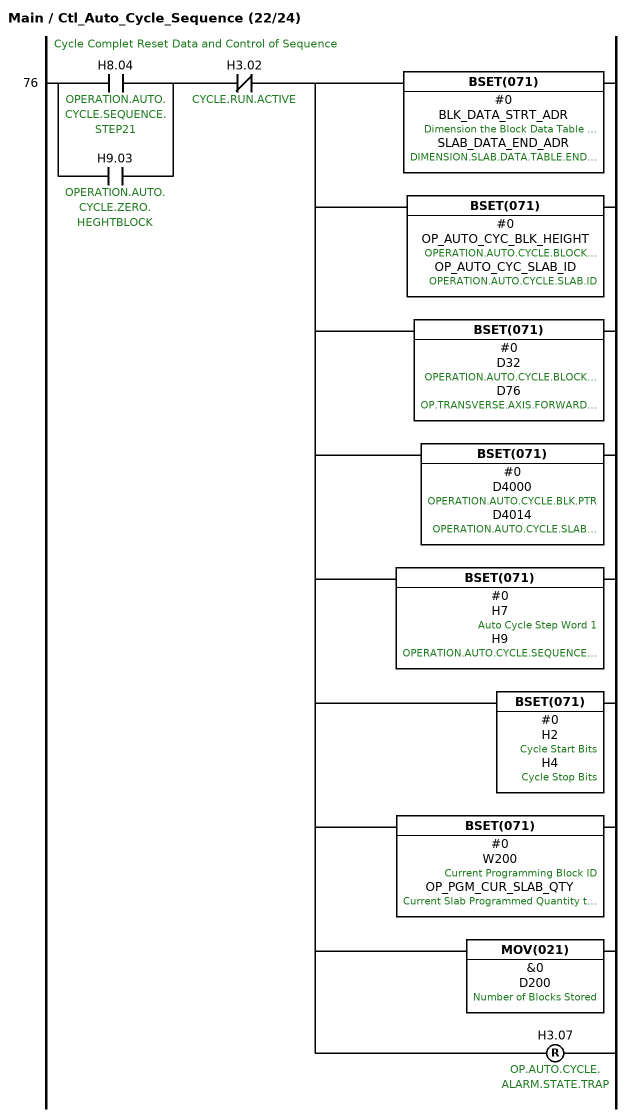
; rung 76: Cycle Complet Reset Data and Control of Sequence
LD H8.04  ; OPERATION.AUTO.CYCLE.SEQUENCE.STEP21
OR H9.03  ; OPERATION.AUTO.CYCLE.ZERO.HEGHTBLOCK
ANDNOT H3.02  ; CYCLE.RUN.ACTIVE
BSET(071) #0 BLK_DATA_STRT_ADR SLAB_DATA_END_ADR  ; Dimension the Block Data Table - Start Address, DIMENSION.SLAB.DATA.TABLE.END.ADDRESS
BSET(071) #0 OP_AUTO_CYC_BLK_HEIGHT OP_AUTO_CYC_SLAB_ID  ; OPERATION.AUTO.CYCLE.BLOCK.HEIGHT.WORKING, OPERATION.AUTO.CYCLE.SLAB.ID
BSET(071) #0 D32 D76  ; OPERATION.AUTO.CYCLE.BLOCK.FIRST.CUT.WORKING.REAL, OP.TRANSVERSE.AXIS.FORWARD.TARGET
BSET(071) #0 D4000 D4014  ; OPERATION.AUTO.CYCLE.BLK.PTR, OPERATION.AUTO.CYCLE.SLAB.POINTER
BSET(071) #0 H7 H9  ; Auto Cycle Step Word 1, OPERATION.AUTO.CYCLE.SEQUENCE.STATE.BITS
BSET(071) #0 H2 H4  ; Cycle Start Bits, Cycle Stop Bits
BSET(071) #0 W200 OP_PGM_CUR_SLAB_QTY  ; Current Programming Block ID, Current Slab Programmed Quantity to cut
MOV(021) &0 D200  ; Number of Blocks Stored
RSET H3.07  ; OP.AUTO.CYCLE.ALARM.STATE.TRAP

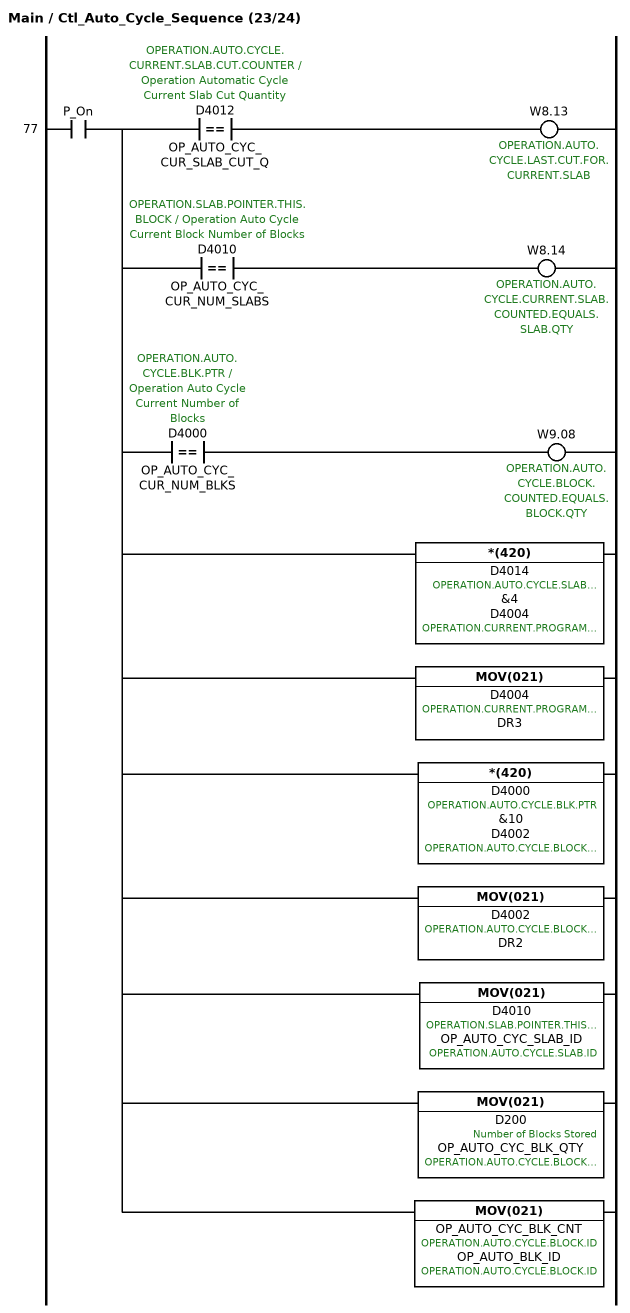
; rung 77
LD P_On
OUT TR0
AND=(300) D4012 OP_AUTO_CYC_CUR_SLAB_CUT_Q  ; OPERATION.AUTO.CYCLE.CURRENT.SLAB.CUT.COUNTER, Operation Automatic Cycle Current Slab Cut Quantity
OUT W8.13  ; OPERATION.AUTO.CYCLE.LAST.CUT.FOR.CURRENT.SLAB
LD TR0
AND=(300) D4010 OP_AUTO_CYC_CUR_NUM_SLABS  ; OPERATION.SLAB.POINTER.THIS.BLOCK, Operation Auto Cycle Current Block Number of Blocks
OUT W8.14  ; OPERATION.AUTO.CYCLE.CURRENT.SLAB.COUNTED.EQUALS.SLAB.QTY
LD TR0
AND=(300) D4000 OP_AUTO_CYC_CUR_NUM_BLKS  ; OPERATION.AUTO.CYCLE.BLK.PTR, Operation Auto Cycle Current Number of Blocks
OUT W9.08  ; OPERATION.AUTO.CYCLE.BLOCK.COUNTED.EQUALS.BLOCK.QTY
LD TR0
*(420) D4014 &4 D4004  ; OPERATION.AUTO.CYCLE.SLAB.POINTER, OPERATION.CURRENT.PROGRAM.SLAB.DATA.POINTER
MOV(021) D4004 DR3  ; OPERATION.CURRENT.PROGRAM.SLAB.DATA.POINTER
*(420) D4000 &10 D4002  ; OPERATION.AUTO.CYCLE.BLK.PTR, OPERATION.AUTO.CYCLE.BLOCK.DATA.POINTER
MOV(021) D4002 DR2  ; OPERATION.AUTO.CYCLE.BLOCK.DATA.POINTER
MOV(021) D4010 OP_AUTO_CYC_SLAB_ID  ; OPERATION.SLAB.POINTER.THIS.BLOCK, OPERATION.AUTO.CYCLE.SLAB.ID
MOV(021) D200 OP_AUTO_CYC_BLK_QTY  ; Number of Blocks Stored, OPERATION.AUTO.CYCLE.BLOCK.QUANTITY
MOV(021) OP_AUTO_CYC_BLK_CNT OP_AUTO_BLK_ID  ; OPERATION.AUTO.CYCLE.BLOCK.ID

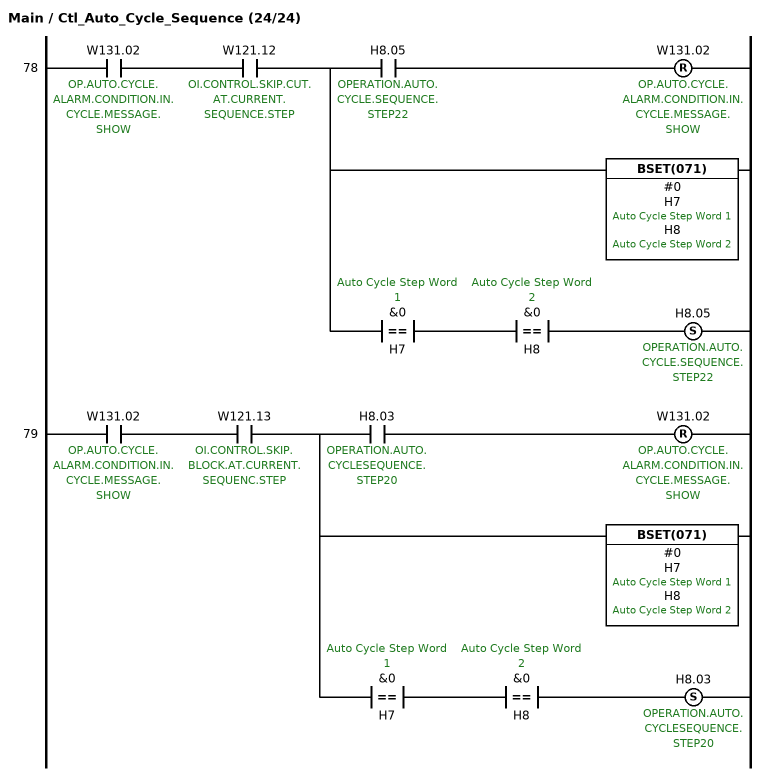
; rung 78
LD W131.02  ; OP.AUTO.CYCLE.ALARM.CONDITION.IN.CYCLE.MESSAGE.SHOW
AND W121.12  ; OI.CONTROL.SKIP.CUT.AT.CURRENT.SEQUENCE.STEP
OUT TR0
AND H8.05  ; OPERATION.AUTO.CYCLE.SEQUENCE.STEP22
RSET W131.02  ; OP.AUTO.CYCLE.ALARM.CONDITION.IN.CYCLE.MESSAGE.SHOW
LD TR0
BSET(071) #0 H7 H8  ; Auto Cycle Step Word 1, Auto Cycle Step Word 2
AND=(300) &0 H7  ; Auto Cycle Step Word 1
AND=(300) &0 H8  ; Auto Cycle Step Word 2
SET H8.05  ; OPERATION.AUTO.CYCLE.SEQUENCE.STEP22
; rung 79
LD W131.02  ; OP.AUTO.CYCLE.ALARM.CONDITION.IN.CYCLE.MESSAGE.SHOW
AND W121.13  ; OI.CONTROL.SKIP.BLOCK.AT.CURRENT.SEQUENC.STEP
OUT TR0
AND H8.03  ; OPERATION.AUTO.CYCLESEQUENCE.STEP20
RSET W131.02  ; OP.AUTO.CYCLE.ALARM.CONDITION.IN.CYCLE.MESSAGE.SHOW
LD TR0
BSET(071) #0 H7 H8  ; Auto Cycle Step Word 1, Auto Cycle Step Word 2
AND=(300) &0 H7  ; Auto Cycle Step Word 1
AND=(300) &0 H8  ; Auto Cycle Step Word 2
SET H8.03  ; OPERATION.AUTO.CYCLESEQUENCE.STEP20

### Section Ctl_Master_Home

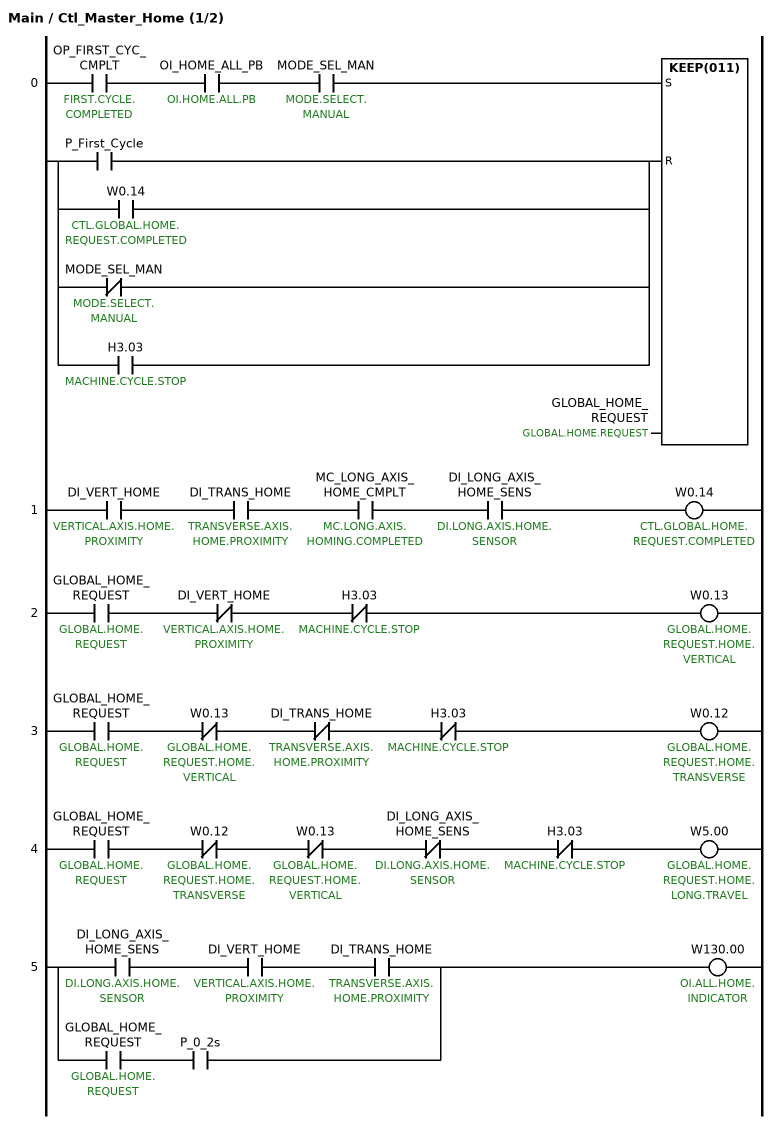
; rung 0
LD OP_FIRST_CYC_CMPLT  ; FIRST.CYCLE.COMPLETED
AND OI_HOME_ALL_PB  ; OI.HOME.ALL.PB
AND MODE_SEL_MAN  ; MODE.SELECT.MANUAL
LD P_First_Cycle
OR W0.14  ; CTL.GLOBAL.HOME.REQUEST.COMPLETED
ORNOT MODE_SEL_MAN  ; MODE.SELECT.MANUAL
OR H3.03  ; MACHINE.CYCLE.STOP
KEEP(011) GLOBAL_HOME_REQUEST  ; GLOBAL.HOME.REQUEST
; rung 1
LD DI_VERT_HOME  ; VERTICAL.AXIS.HOME.PROXIMITY
AND DI_TRANS_HOME  ; TRANSVERSE.AXIS.HOME.PROXIMITY
AND MC_LONG_AXIS_HOME_CMPLT  ; MC.LONG.AXIS.HOMING.COMPLETED
AND DI_LONG_AXIS_HOME_SENS  ; DI.LONG.AXIS.HOME.SENSOR
OUT W0.14  ; CTL.GLOBAL.HOME.REQUEST.COMPLETED
; rung 2
LD GLOBAL_HOME_REQUEST  ; GLOBAL.HOME.REQUEST
ANDNOT DI_VERT_HOME  ; VERTICAL.AXIS.HOME.PROXIMITY
ANDNOT H3.03  ; MACHINE.CYCLE.STOP
OUT W0.13  ; GLOBAL.HOME.REQUEST.HOME.VERTICAL
; rung 3
LD GLOBAL_HOME_REQUEST  ; GLOBAL.HOME.REQUEST
ANDNOT W0.13  ; GLOBAL.HOME.REQUEST.HOME.VERTICAL
ANDNOT DI_TRANS_HOME  ; TRANSVERSE.AXIS.HOME.PROXIMITY
ANDNOT H3.03  ; MACHINE.CYCLE.STOP
OUT W0.12  ; GLOBAL.HOME.REQUEST.HOME.TRANSVERSE
; rung 4
LD GLOBAL_HOME_REQUEST  ; GLOBAL.HOME.REQUEST
ANDNOT W0.12  ; GLOBAL.HOME.REQUEST.HOME.TRANSVERSE
ANDNOT W0.13  ; GLOBAL.HOME.REQUEST.HOME.VERTICAL
ANDNOT DI_LONG_AXIS_HOME_SENS  ; DI.LONG.AXIS.HOME.SENSOR
ANDNOT H3.03  ; MACHINE.CYCLE.STOP
OUT W5.00  ; GLOBAL.HOME.REQUEST.HOME.LONG.TRAVEL
; rung 5
LD DI_LONG_AXIS_HOME_SENS  ; DI.LONG.AXIS.HOME.SENSOR
AND DI_VERT_HOME  ; VERTICAL.AXIS.HOME.PROXIMITY
AND DI_TRANS_HOME  ; TRANSVERSE.AXIS.HOME.PROXIMITY
LD GLOBAL_HOME_REQUEST  ; GLOBAL.HOME.REQUEST
AND P_0_2s
ORLD
OUT W130.00  ; OI.ALL.HOME.INDICATOR

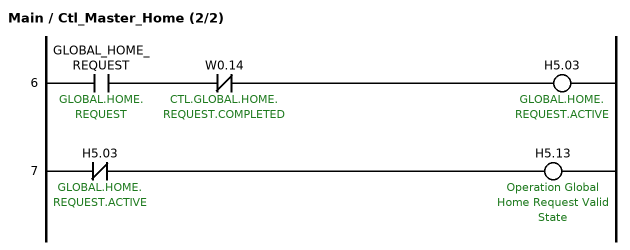
; rung 6
LD GLOBAL_HOME_REQUEST  ; GLOBAL.HOME.REQUEST
ANDNOT W0.14  ; CTL.GLOBAL.HOME.REQUEST.COMPLETED
OUT H5.03  ; GLOBAL.HOME.REQUEST.ACTIVE
; rung 7
LDNOT H5.03  ; GLOBAL.HOME.REQUEST.ACTIVE
OUT H5.13  ; Operation Global Home Request Valid State

### Section Ctl_Long_Axis

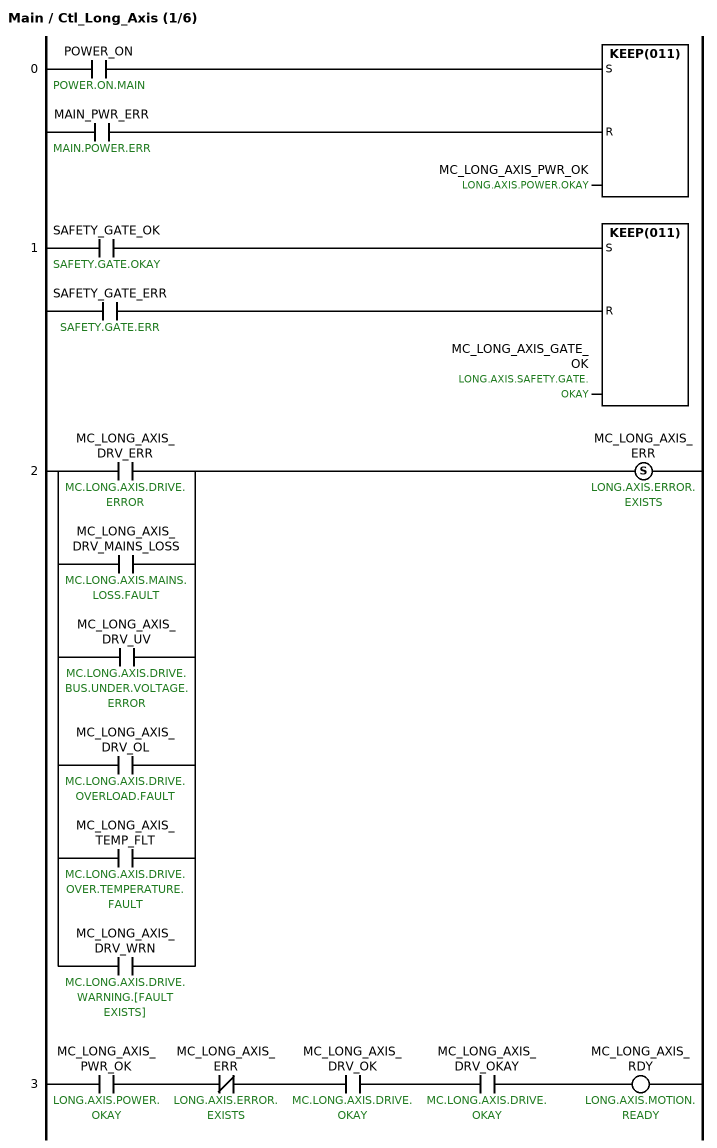
; rung 0
LD POWER_ON  ; POWER.ON.MAIN
LD MAIN_PWR_ERR  ; MAIN.POWER.ERR
KEEP(011) MC_LONG_AXIS_PWR_OK  ; LONG.AXIS.POWER.OKAY
; rung 1
LD SAFETY_GATE_OK  ; SAFETY.GATE.OKAY
LD SAFETY_GATE_ERR  ; SAFETY.GATE.ERR
KEEP(011) MC_LONG_AXIS_GATE_OK  ; LONG.AXIS.SAFETY.GATE.OKAY
; rung 2
LD MC_LONG_AXIS_DRV_ERR  ; MC.LONG.AXIS.DRIVE.ERROR
OR MC_LONG_AXIS_DRV_MAINS_LOSS  ; MC.LONG.AXIS.MAINS.LOSS.FAULT
OR MC_LONG_AXIS_DRV_UV  ; MC.LONG.AXIS.DRIVE.BUS.UNDER.VOLTAGE.ERROR
OR MC_LONG_AXIS_DRV_OL  ; MC.LONG.AXIS.DRIVE.OVERLOAD.FAULT
OR MC_LONG_AXIS_TEMP_FLT  ; MC.LONG.AXIS.DRIVE.OVER.TEMPERATURE.FAULT
OR MC_LONG_AXIS_DRV_WRN  ; MC.LONG.AXIS.DRIVE.WARNING.[FAULT EXISTS]
SET MC_LONG_AXIS_ERR  ; LONG.AXIS.ERROR.EXISTS
; rung 3
LD MC_LONG_AXIS_PWR_OK  ; LONG.AXIS.POWER.OKAY
ANDNOT MC_LONG_AXIS_ERR  ; LONG.AXIS.ERROR.EXISTS
AND MC_LONG_AXIS_DRV_OK  ; MC.LONG.AXIS.DRIVE.OKAY
AND MC_LONG_AXIS_DRV_OKAY  ; MC.LONG.AXIS.DRIVE.OKAY
OUT MC_LONG_AXIS_RDY  ; LONG.AXIS.MOTION.READY

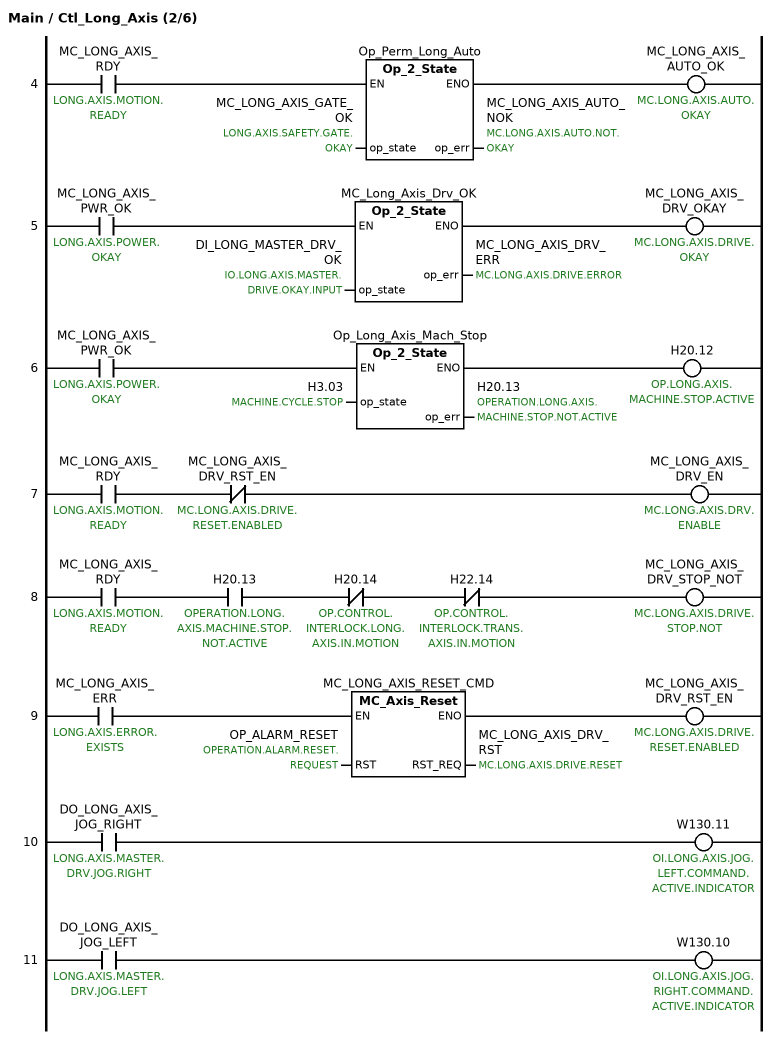
; rung 4
LD MC_LONG_AXIS_RDY  ; LONG.AXIS.MOTION.READY
CALL Op_Perm_Long_Auto : Op_2_State (op_state := MC_LONG_AXIS_GATE_OK, op_err => MC_LONG_AXIS_AUTO_NOK)  ; LONG.AXIS.SAFETY.GATE.OKAY, MC.LONG.AXIS.AUTO.NOT.OKAY
OUT MC_LONG_AXIS_AUTO_OK  ; MC.LONG.AXIS.AUTO.OKAY
; rung 5
LD MC_LONG_AXIS_PWR_OK  ; LONG.AXIS.POWER.OKAY
CALL MC_Long_Axis_Drv_OK : Op_2_State (op_state := DI_LONG_MASTER_DRV_OK, op_err => MC_LONG_AXIS_DRV_ERR)  ; IO.LONG.AXIS.MASTER.DRIVE.OKAY.INPUT, MC.LONG.AXIS.DRIVE.ERROR
OUT MC_LONG_AXIS_DRV_OKAY  ; MC.LONG.AXIS.DRIVE.OKAY
; rung 6
LD MC_LONG_AXIS_PWR_OK  ; LONG.AXIS.POWER.OKAY
CALL Op_Long_Axis_Mach_Stop : Op_2_State (op_state := H3.03, op_err => H20.13)  ; MACHINE.CYCLE.STOP, OPERATION.LONG.AXIS.MACHINE.STOP.NOT.ACTIVE
OUT H20.12  ; OP.LONG.AXIS.MACHINE.STOP.ACTIVE
; rung 7
LD MC_LONG_AXIS_RDY  ; LONG.AXIS.MOTION.READY
ANDNOT MC_LONG_AXIS_DRV_RST_EN  ; MC.LONG.AXIS.DRIVE.RESET.ENABLED
OUT MC_LONG_AXIS_DRV_EN  ; MC.LONG.AXIS.DRV.ENABLE
; rung 8
LD MC_LONG_AXIS_RDY  ; LONG.AXIS.MOTION.READY
AND H20.13  ; OPERATION.LONG.AXIS.MACHINE.STOP.NOT.ACTIVE
ANDNOT H20.14  ; OP.CONTROL.INTERLOCK.LONG.AXIS.IN.MOTION
ANDNOT H22.14  ; OP.CONTROL.INTERLOCK.TRANS.AXIS.IN.MOTION
OUT MC_LONG_AXIS_DRV_STOP_NOT  ; MC.LONG.AXIS.DRIVE.STOP.NOT
; rung 9
LD MC_LONG_AXIS_ERR  ; LONG.AXIS.ERROR.EXISTS
CALL MC_LONG_AXIS_RESET_CMD : MC_Axis_Reset (RST := OP_ALARM_RESET, RST_REQ => MC_LONG_AXIS_DRV_RST)  ; OPERATION.ALARM.RESET.REQUEST, MC.LONG.AXIS.DRIVE.RESET
OUT MC_LONG_AXIS_DRV_RST_EN  ; MC.LONG.AXIS.DRIVE.RESET.ENABLED
; rung 10
LD DO_LONG_AXIS_JOG_RIGHT  ; LONG.AXIS.MASTER.DRV.JOG.RIGHT
OUT W130.11  ; OI.LONG.AXIS.JOG.LEFT.COMMAND.ACTIVE.INDICATOR
; rung 11
LD DO_LONG_AXIS_JOG_LEFT  ; LONG.AXIS.MASTER.DRV.JOG.LEFT
OUT W130.10  ; OI.LONG.AXIS.JOG.RIGHT.COMMAND.ACTIVE.INDICATOR

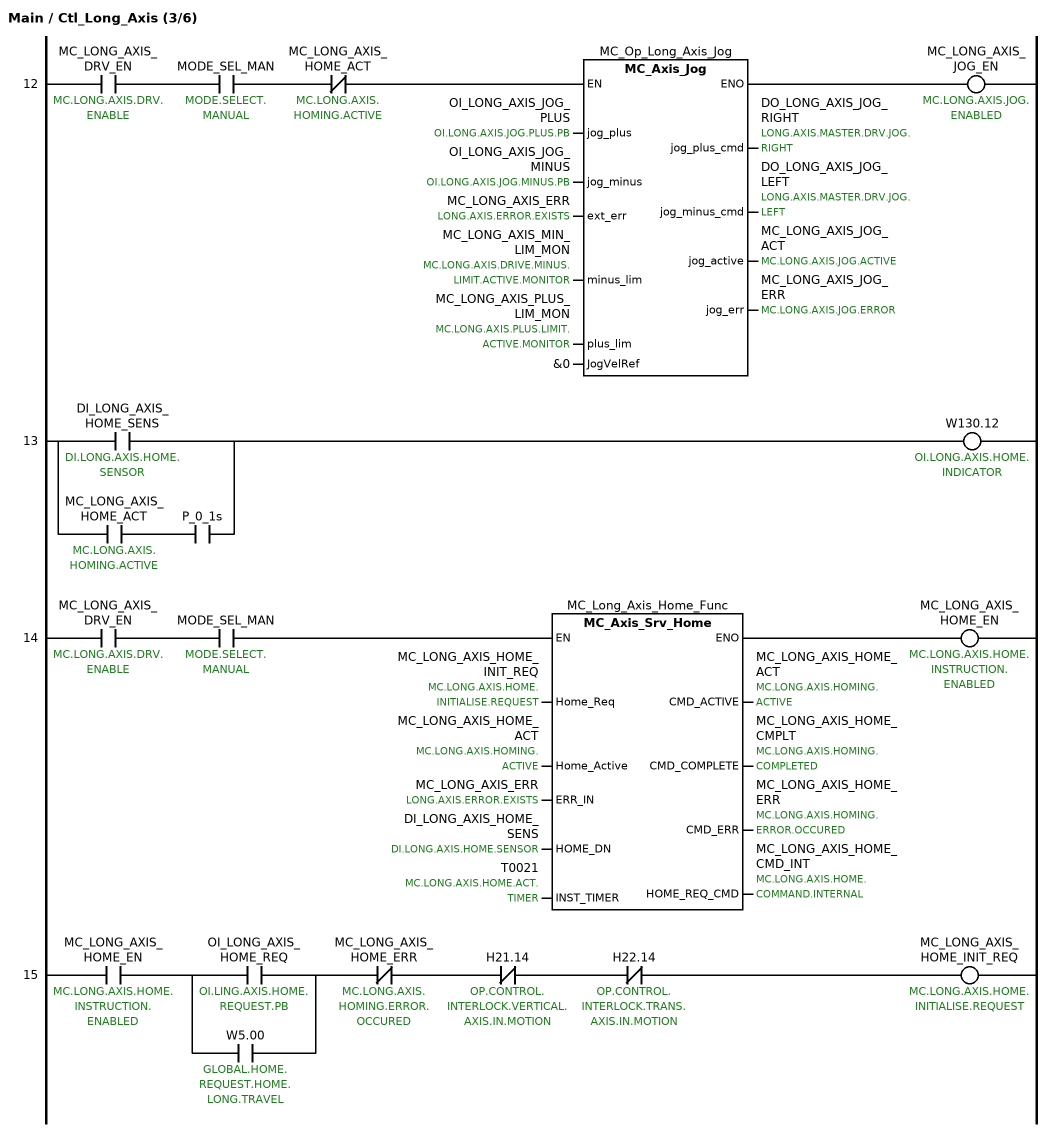
; rung 12
LD MC_LONG_AXIS_DRV_EN  ; MC.LONG.AXIS.DRV.ENABLE
AND MODE_SEL_MAN  ; MODE.SELECT.MANUAL
ANDNOT MC_LONG_AXIS_HOME_ACT  ; MC.LONG.AXIS.HOMING.ACTIVE
CALL MC_Op_Long_Axis_Jog : MC_Axis_Jog (jog_plus := OI_LONG_AXIS_JOG_PLUS, jog_minus := OI_LONG_AXIS_JOG_MINUS, ext_err := MC_LONG_AXIS_ERR, minus_lim := MC_LONG_AXIS_MIN_LIM_MON, plus_lim := MC_LONG_AXIS_PLUS_LIM_MON, JogVelRef := &0, jog_plus_cmd => DO_LONG_AXIS_JOG_RIGHT, jog_minus_cmd => DO_LONG_AXIS_JOG_LEFT, jog_active => MC_LONG_AXIS_JOG_ACT, jog_err => MC_LONG_AXIS_JOG_ERR)  ; OI.LONG.AXIS.JOG.PLUS.PB, OI.LONG.AXIS.JOG.MINUS.PB, LONG.AXIS.ERROR.EXISTS, MC.LONG.AXIS.DRIVE.MINUS.LIMIT.ACTIVE.MONITOR, MC.LONG.AXIS.PLUS.LIMIT.ACTIVE.MONITOR, LONG.AXIS.MASTER.DRV.JOG.RIGHT, LONG.AXIS.MASTER.DRV.JOG.LEFT, MC.LONG.AXIS.JOG.ACTIVE, MC.LONG.AXIS.JOG.ERROR
OUT MC_LONG_AXIS_JOG_EN  ; MC.LONG.AXIS.JOG.ENABLED
; rung 13
LD DI_LONG_AXIS_HOME_SENS  ; DI.LONG.AXIS.HOME.SENSOR
LD MC_LONG_AXIS_HOME_ACT  ; MC.LONG.AXIS.HOMING.ACTIVE
AND P_0_1s
ORLD
OUT W130.12  ; OI.LONG.AXIS.HOME.INDICATOR
; rung 14
LD MC_LONG_AXIS_DRV_EN  ; MC.LONG.AXIS.DRV.ENABLE
AND MODE_SEL_MAN  ; MODE.SELECT.MANUAL
CALL MC_Long_Axis_Home_Func : MC_Axis_Srv_Home (Home_Req := MC_LONG_AXIS_HOME_INIT_REQ, Home_Active := MC_LONG_AXIS_HOME_ACT, ERR_IN := MC_LONG_AXIS_ERR, HOME_DN := DI_LONG_AXIS_HOME_SENS, INST_TIMER := T0021, CMD_ACTIVE => MC_LONG_AXIS_HOME_ACT, CMD_COMPLETE => MC_LONG_AXIS_HOME_CMPLT, CMD_ERR => MC_LONG_AXIS_HOME_ERR, HOME_REQ_CMD => MC_LONG_AXIS_HOME_CMD_INT)  ; MC.LONG.AXIS.HOME.INITIALISE.REQUEST, MC.LONG.AXIS.HOMING.ACTIVE, LONG.AXIS.ERROR.EXISTS, DI.LONG.AXIS.HOME.SENSOR, MC.LONG.AXIS.HOME.ACT.TIMER, MC.LONG.AXIS.HOMING.COMPLETED, MC.LONG.AXIS.HOMING.ERROR.OCCURED, MC.LONG.AXIS.HOME.COMMAND.INTERNAL
OUT MC_LONG_AXIS_HOME_EN  ; MC.LONG.AXIS.HOME.INSTRUCTION.ENABLED
; rung 15
LD MC_LONG_AXIS_HOME_EN  ; MC.LONG.AXIS.HOME.INSTRUCTION.ENABLED
LD OI_LONG_AXIS_HOME_REQ  ; OI.LING.AXIS.HOME.REQUEST.PB
OR W5.00  ; GLOBAL.HOME.REQUEST.HOME.LONG.TRAVEL
ANDLD
ANDNOT MC_LONG_AXIS_HOME_ERR  ; MC.LONG.AXIS.HOMING.ERROR.OCCURED
ANDNOT H21.14  ; OP.CONTROL.INTERLOCK.VERTICAL.AXIS.IN.MOTION
ANDNOT H22.14  ; OP.CONTROL.INTERLOCK.TRANS.AXIS.IN.MOTION
OUT MC_LONG_AXIS_HOME_INIT_REQ  ; MC.LONG.AXIS.HOME.INITIALISE.REQUEST

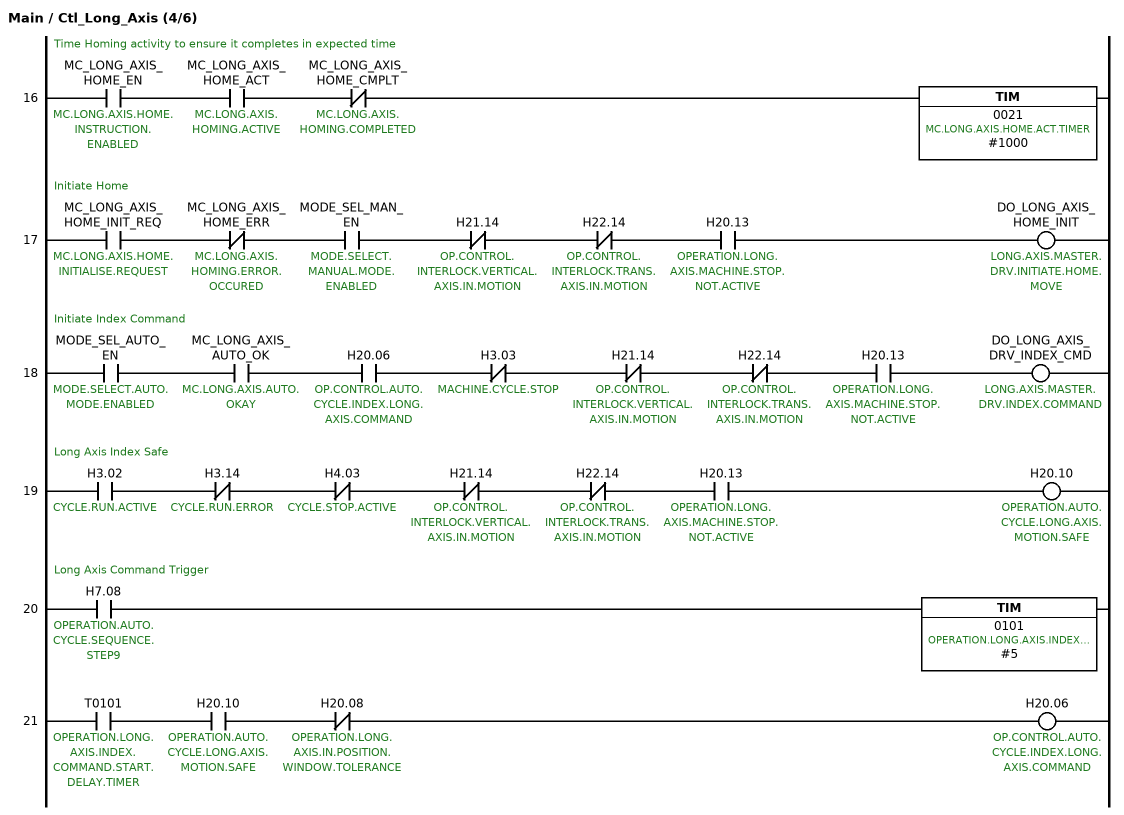
; rung 16: Time Homing activity to ensure it completes in expected time
LD MC_LONG_AXIS_HOME_EN  ; MC.LONG.AXIS.HOME.INSTRUCTION.ENABLED
AND MC_LONG_AXIS_HOME_ACT  ; MC.LONG.AXIS.HOMING.ACTIVE
ANDNOT MC_LONG_AXIS_HOME_CMPLT  ; MC.LONG.AXIS.HOMING.COMPLETED
TIM 0021 #1000  ; MC.LONG.AXIS.HOME.ACT.TIMER
; rung 17: Initiate Home
LD MC_LONG_AXIS_HOME_INIT_REQ  ; MC.LONG.AXIS.HOME.INITIALISE.REQUEST
ANDNOT MC_LONG_AXIS_HOME_ERR  ; MC.LONG.AXIS.HOMING.ERROR.OCCURED
AND MODE_SEL_MAN_EN  ; MODE.SELECT.MANUAL.MODE.ENABLED
ANDNOT H21.14  ; OP.CONTROL.INTERLOCK.VERTICAL.AXIS.IN.MOTION
ANDNOT H22.14  ; OP.CONTROL.INTERLOCK.TRANS.AXIS.IN.MOTION
AND H20.13  ; OPERATION.LONG.AXIS.MACHINE.STOP.NOT.ACTIVE
OUT DO_LONG_AXIS_HOME_INIT  ; LONG.AXIS.MASTER.DRV.INITIATE.HOME.MOVE
; rung 18: Initiate Index Command
LD MODE_SEL_AUTO_EN  ; MODE.SELECT.AUTO.MODE.ENABLED
AND MC_LONG_AXIS_AUTO_OK  ; MC.LONG.AXIS.AUTO.OKAY
AND H20.06  ; OP.CONTROL.AUTO.CYCLE.INDEX.LONG.AXIS.COMMAND
ANDNOT H3.03  ; MACHINE.CYCLE.STOP
ANDNOT H21.14  ; OP.CONTROL.INTERLOCK.VERTICAL.AXIS.IN.MOTION
ANDNOT H22.14  ; OP.CONTROL.INTERLOCK.TRANS.AXIS.IN.MOTION
AND H20.13  ; OPERATION.LONG.AXIS.MACHINE.STOP.NOT.ACTIVE
OUT DO_LONG_AXIS_DRV_INDEX_CMD  ; LONG.AXIS.MASTER.DRV.INDEX.COMMAND
; rung 19: Long Axis Index Safe
LD H3.02  ; CYCLE.RUN.ACTIVE
ANDNOT H3.14  ; CYCLE.RUN.ERROR
ANDNOT H4.03  ; CYCLE.STOP.ACTIVE
ANDNOT H21.14  ; OP.CONTROL.INTERLOCK.VERTICAL.AXIS.IN.MOTION
ANDNOT H22.14  ; OP.CONTROL.INTERLOCK.TRANS.AXIS.IN.MOTION
AND H20.13  ; OPERATION.LONG.AXIS.MACHINE.STOP.NOT.ACTIVE
OUT H20.10  ; OPERATION.AUTO.CYCLE.LONG.AXIS.MOTION.SAFE
; rung 20: Long Axis Command Trigger
LD H7.08  ; OPERATION.AUTO.CYCLE.SEQUENCE.STEP9
TIM 0101 #5  ; OPERATION.LONG.AXIS.INDEX.COMMAND.START.DELAY.TIMER
; rung 21
LD T0101  ; OPERATION.LONG.AXIS.INDEX.COMMAND.START.DELAY.TIMER
AND H20.10  ; OPERATION.AUTO.CYCLE.LONG.AXIS.MOTION.SAFE
ANDNOT H20.08  ; OPERATION.LONG.AXIS.IN.POSITION.WINDOW.TOLERANCE
OUT H20.06  ; OP.CONTROL.AUTO.CYCLE.INDEX.LONG.AXIS.COMMAND

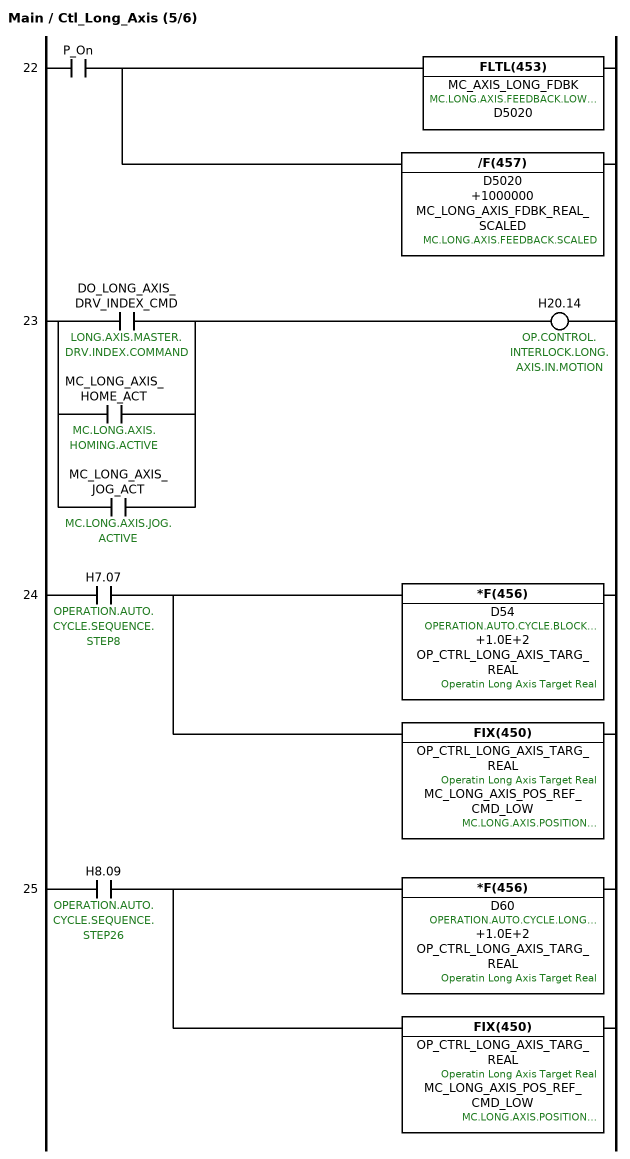
; rung 22
LD P_On
FLTL(453) MC_AXIS_LONG_FDBK D5020  ; MC.LONG.AXIS.FEEDBACK.LOW.WORD
/F(457) D5020 +1000000 MC_LONG_AXIS_FDBK_REAL_SCALED  ; MC.LONG.AXIS.FEEDBACK.SCALED
; rung 23
LD DO_LONG_AXIS_DRV_INDEX_CMD  ; LONG.AXIS.MASTER.DRV.INDEX.COMMAND
OR MC_LONG_AXIS_HOME_ACT  ; MC.LONG.AXIS.HOMING.ACTIVE
OR MC_LONG_AXIS_JOG_ACT  ; MC.LONG.AXIS.JOG.ACTIVE
OUT H20.14  ; OP.CONTROL.INTERLOCK.LONG.AXIS.IN.MOTION
; rung 24
LD H7.07  ; OPERATION.AUTO.CYCLE.SEQUENCE.STEP8
*F(456) D54 +1.0E+2 OP_CTRL_LONG_AXIS_TARG_REAL  ; OPERATION.AUTO.CYCLE.BLOCK.FIRST.CUT.REAL, Operatin Long Axis Target Real
FIX(450) OP_CTRL_LONG_AXIS_TARG_REAL MC_LONG_AXIS_POS_REF_CMD_LOW  ; Operatin Long Axis Target Real, MC.LONG.AXIS.POSITION.REFERENCE.COMMAND.VALUE.LOW.WORD
; rung 25
LD H8.09  ; OPERATION.AUTO.CYCLE.SEQUENCE.STEP26
*F(456) D60 +1.0E+2 OP_CTRL_LONG_AXIS_TARG_REAL  ; OPERATION.AUTO.CYCLE.LONG.INDEX.LOCATION.REAL, Operatin Long Axis Target Real
FIX(450) OP_CTRL_LONG_AXIS_TARG_REAL MC_LONG_AXIS_POS_REF_CMD_LOW  ; Operatin Long Axis Target Real, MC.LONG.AXIS.POSITION.REFERENCE.COMMAND.VALUE.LOW.WORD

